C05485=1219.742,-85.560,-37.736,179.582,5.371,149.062
C05486=1219.736,-85.310,-37.746,179.584,5.371,149.061
C05487=1219.731,-85.061,-37.758,179.587,5.372,149.061
C05488=1219.726,-84.810,-37.768,179.589,5.371,149.060
C05489=1219.721,-84.561,-37.779,179.592,5.372,149.059
C05490=1219.715,-84.311,-37.790,179.594,5.371,149.058
C05491=1219.711,-84.061,-37.802,179.596,5.372,149.058
C05492=1219.705,-83.812,-37.813,179.599,5.372,149.057
C05493=1219.700,-83.562,-37.823,179.601,5.372,149.056
C05494=1219.696,-83.312,-37.834,179.603,5.372,149.056
C05495=1219.689,-83.063,-37.845,179.606,5.372,149.055
C05496=1219.685,-82.813,-37.857,179.608,5.372,149.054
C05497=1219.680,-82.563,-37.868,179.610,5.373,149.054
C05498=1219.674,-82.314,-37.878,179.612,5.372,149.053
C05499=1219.669,-82.064,-37.890,179.615,5.373,149.052
C05500=1219.664,-81.814,-37.901,179.617,5.372,149.052
C05501=1219.659,-81.565,-37.911,179.620,5.373,149.051
C05502=1219.653,-81.315,-37.923,179.622,5.372,149.050
C05503=1219.648,-81.064,-37.934,179.625,5.373,149.049
C05504=1219.643,-80.816,-37.945,179.627,5.372,149.049
C05505=1219.638,-80.566,-37.956,179.629,5.373,149.048
C05506=1219.632,-80.315,-37.967,179.632,5.374,149.048
C05507=1219.627,-80.066,-37.978,179.634,5.373,149.047
C05508=1219.622,-79.817,-37.990,179.636,5.374,149.046
C05509=1219.617,-79.567,-38.001,179.638,5.373,149.045
C05510=1219.612,-79.317,-38.012,179.641,5.374,149.045
C05511=1219.607,-79.068,-38.023,179.643,5.374,149.044
C05512=1219.601,-78.818,-38.035,179.646,5.374,149.043
C05513=1219.596,-78.568,-38.045,179.648,5.374,149.043
C05514=1219.591,-78.319,-38.056,179.651,5.374,149.042
C05515=1219.586,-78.069,-38.068,179.653,5.374,149.041
C05516=1219.581,-77.819,-38.079,179.655,5.374,149.041
C05517=1219.576,-77.569,-38.090,179.657,5.374,149.040
C05518=1219.570,-77.320,-38.102,179.660,5.375,149.039
C05519=1219.565,-77.070,-38.113,179.662,5.374,149.039
C05520=1219.561,-76.820,-38.124,179.664,5.375,149.038
C05521=1219.554,-76.571,-38.136,179.667,5.375,149.037
C05522=1219.549,-76.321,-38.146,179.669,5.375,149.036
C05523=1219.544,-76.071,-38.158,179.672,5.375,149.036
C05524=1219.539,-75.821,-38.169,179.674,5.375,149.035
C05525=1219.534,-75.572,-38.180,179.677,5.375,149.034
C05526=1219.529,-75.322,-38.192,179.679,5.375,149.034
C05527=1219.523,-75.051,-38.204,179.681,5.375,149.033
C05528=1219.517,-74.781,-38.216,179.684,5.376,149.032
C05529=1219.512,-74.511,-38.229,179.686,5.376,149.032
C05530=1219.507,-74.240,-38.241,179.689,5.376,149.031
C05531=1219.501,-73.991,-38.253,179.691,5.376,149.030
C05532=1219.496,-73.741,-38.264,179.693,5.376,149.029
C05533=1219.490,-73.491,-38.276,179.696,5.377,149.029
C05534=1219.485,-73.241,-38.286,179.698,5.376,149.028
C05535=1219.480,-72.991,-38.298,179.701,5.377,149.027
C05536=1219.475,-72.742,-38.309,179.703,5.376,149.027
C05537=1219.470,-72.493,-38.320,179.706,5.377,149.026
C05538=1219.465,-72.243,-38.332,179.708,5.376,149.025
C05539=1219.460,-71.993,-38.344,179.710,5.377,149.024
C05540=1219.454,-71.743,-38.355,179.713,5.377,149.024
C05541=1219.449,-71.494,-38.366,179.715,5.377,149.023
C05542=1219.444,-71.244,-38.378,179.718,5.377,149.022
C05543=1219.439,-70.995,-38.390,179.720,5.377,149.022
C05544=1219.434,-70.745,-38.401,179.723,5.378,149.021
C05545=1219.429,-70.495,-38.413,179.724,5.378,149.020
C05546=1219.423,-70.246,-38.424,179.727,5.378,149.020
C05547=1219.418,-69.996,-38.435,179.729,5.378,149.019
C05548=1219.413,-69.746,-38.447,179.732,5.378,149.018
C05549=1219.408,-69.496,-38.458,179.734,5.378,149.018
C05550=1219.402,-69.246,-38.470,179.736,5.378,149.017
C05551=1219.398,-68.996,-38.481,179.739,5.379,149.016
C05552=1219.392,-68.747,-38.493,179.741,5.378,149.015
C05553=1219.386,-68.497,-38.505,179.744,5.379,149.015
C05554=1219.382,-68.248,-38.516,179.746,5.378,149.014
C05555=1219.376,-67.998,-38.528,179.749,5.379,149.013
C05556=1219.372,-67.749,-38.540,179.751,5.379,149.013
C05557=1219.366,-67.499,-38.552,179.753,5.379,149.012
C05558=1219.362,-67.249,-38.563,179.755,5.379,149.011
C05559=1219.356,-67.000,-38.574,179.758,5.379,149.011
C05560=1219.351,-66.750,-38.586,179.760,5.380,149.010
C05561=1219.345,-66.500,-38.598,179.762,5.380,149.009
C05562=1219.340,-66.250,-38.609,179.765,5.380,149.009
C05563=1219.335,-66.001,-38.621,179.767,5.380,149.008
C05564=1219.330,-65.751,-38.633,179.770,5.380,149.007
C05565=1219.325,-65.501,-38.644,179.772,5.380,149.007
C05566=1219.320,-65.251,-38.656,179.775,5.380,149.006
C05567=1219.314,-65.001,-38.668,179.777,5.381,149.005
C05568=1219.309,-64.752,-38.679,179.779,5.380,149.004
C05569=1219.304,-64.503,-38.691,179.782,5.381,149.004
C05570=1219.299,-64.254,-38.703,179.784,5.381,149.003
C05571=1219.294,-64.004,-38.714,179.787,5.381,149.002
C05572=1219.288,-63.754,-38.726,179.789,5.381,149.002
C05573=1219.284,-63.504,-38.738,179.791,5.381,149.001
C05574=1219.278,-63.254,-38.749,179.794,5.382,149.000
C05575=1219.273,-63.005,-38.762,179.796,5.381,148.999
C05576=1219.268,-62.755,-38.773,179.799,5.382,148.999
C05577=1219.263,-62.505,-38.785,179.801,5.381,148.998
C05578=1219.258,-62.255,-38.797,179.803,5.382,148.998
C05579=1219.253,-62.006,-38.808,179.805,5.382,148.997
C05580=1219.247,-61.756,-38.820,179.808,5.382,148.996
C05581=1219.242,-61.507,-38.833,179.811,5.383,148.995
C05582=1219.237,-61.257,-38.844,179.813,5.382,148.995
C05583=1219.232,-61.008,-38.856,179.815,5.383,148.994
C05584=1219.226,-60.758,-38.868,179.817,5.383,148.993
C05585=1219.222,-60.509,-38.880,179.820,5.383,148.993
C05586=1219.216,-60.259,-38.891,179.822,5.383,148.992
C05587=1219.211,-60.009,-38.903,179.825,5.383,148.991
C05588=1219.206,-59.759,-38.915,179.828,5.384,148.991
C05589=1219.201,-59.510,-38.927,179.830,5.383,148.990
C05590=1219.196,-59.260,-38.939,179.832,5.384,148.989
C05591=1219.190,-59.010,-38.951,179.834,5.383,148.988
C05592=1219.186,-58.761,-38.963,179.837,5.384,148.988
C05593=1219.180,-58.511,-38.975,179.840,5.384,148.987
C05594=1219.175,-58.261,-38.987,179.842,5.384,148.986
C05595=1219.170,-58.011,-38.999,179.844,5.384,148.986
C05596=1219.165,-57.762,-39.011,179.847,5.384,148.985
C05597=1219.160,-57.512,-39.023,179.849,5.385,148.984
C05598=1219.154,-57.262,-39.034,179.851,5.385,148.984
C05599=1219.149,-57.013,-39.047,179.853,5.385,148.983
C05600=1219.145,-56.763,-39.058,179.856,5.385,148.982
C05601=1219.139,-56.514,-39.071,179.858,5.385,148.982
C05602=1219.134,-56.264,-39.083,179.861,5.386,148.981
C05603=1219.129,-56.014,-39.095,179.863,5.385,148.980
C05604=1219.123,-55.765,-39.107,179.866,5.386,148.979
C05605=1219.119,-55.515,-39.119,179.868,5.386,148.979
C05606=1219.113,-55.265,-39.131,179.870,5.386,148.978
C05607=1219.108,-55.016,-39.143,179.873,5.386,148.977
C05608=1219.103,-54.766,-39.155,179.875,5.386,148.977
C05609=1219.098,-54.517,-39.168,179.878,5.386,148.976
C05610=1219.093,-54.267,-39.179,179.880,5.387,148.975
C05611=1219.088,-54.016,-39.191,179.883,5.387,148.975
C05612=1219.083,-53.767,-39.204,179.885,5.387,148.974
C05613=1219.078,-53.517,-39.216,179.887,5.387,148.973
C05614=1219.072,-53.268,-39.228,179.890,5.387,148.972
C05615=1219.067,-53.018,-39.240,179.893,5.388,148.972
C05616=1219.063,-52.769,-39.252,179.895,5.387,148.971
C05617=1219.057,-52.519,-39.264,179.897,5.388,148.970
C05618=1219.052,-52.270,-39.277,179.899,5.387,148.970
C05619=1219.047,-52.020,-39.288,179.902,5.388,148.969
C05620=1219.042,-51.770,-39.301,179.904,5.389,148.968
C05621=1219.036,-51.520,-39.313,179.906,5.388,148.968
C05622=1219.031,-51.271,-39.326,179.909,5.389,148.967
C05623=1219.026,-51.021,-39.337,179.911,5.389,148.966
C05624=1219.021,-50.772,-39.349,179.914,5.389,148.966
C05625=1219.016,-50.521,-39.362,179.916,5.389,148.965
C05626=1219.011,-50.272,-39.374,179.919,5.389,148.964
C05627=1219.006,-50.022,-39.386,179.921,5.390,148.964
C05628=1219.001,-49.773,-39.399,179.924,5.390,148.963
C05629=1218.995,-49.523,-39.411,179.926,5.390,148.962
C05630=1218.990,-49.274,-39.423,179.929,5.390,148.961
C05631=1218.985,-49.003,-39.436,179.931,5.390,148.961
C05632=1218.979,-48.734,-39.450,179.933,5.390,148.960
C05633=1218.973,-48.464,-39.463,179.937,5.390,148.959
C05634=1218.968,-48.194,-39.477,179.939,5.391,148.958
C05635=1218.963,-47.944,-39.489,179.941,5.391,148.958
C05636=1218.958,-47.695,-39.501,179.944,5.391,148.957
C05637=1218.952,-47.445,-39.514,179.947,5.392,148.956
C05638=1218.947,-47.195,-39.526,179.949,5.391,148.956
C05639=1218.942,-46.946,-39.538,179.951,5.392,148.955
C05640=1218.937,-46.696,-39.551,179.953,5.391,148.954
C05641=1218.932,-46.446,-39.563,179.956,5.392,148.953
C05642=1218.927,-46.197,-39.576,179.959,5.392,148.953
C05643=1218.922,-45.947,-39.588,179.960,5.392,148.952
C05644=1218.916,-45.698,-39.600,179.963,5.393,148.952
C05645=1218.911,-45.448,-39.613,179.966,5.393,148.951
C05646=1218.906,-45.199,-39.626,179.968,5.393,148.950
C05647=1218.901,-44.948,-39.638,179.970,5.393,148.949
C05648=1218.896,-44.699,-39.650,179.973,5.393,148.949
C05649=1218.891,-44.450,-39.663,179.975,5.394,148.948
C05650=1218.886,-44.200,-39.675,179.978,5.394,148.947
C05651=1218.880,-43.950,-39.687,179.980,5.394,148.947
C05652=1218.876,-43.700,-39.700,179.983,5.394,148.946
C05653=1218.871,-43.451,-39.713,179.985,5.395,148.945
C05654=1218.865,-43.201,-39.725,179.987,5.394,148.945
C05655=1218.860,-42.952,-39.738,179.990,5.395,148.944
C05656=1218.855,-42.702,-39.750,179.992,5.394,148.943
C05657=1218.851,-42.452,-39.763,179.995,5.395,148.942
C05658=1218.845,-42.203,-39.775,179.997,5.395,148.942
C05659=1218.839,-41.953,-39.788,180.000,5.395,148.941
C05660=1218.834,-41.704,-39.801,-179.998,5.396,148.940
C05661=1218.829,-41.454,-39.813,-179.995,5.396,148.940
C05662=1218.824,-41.204,-39.826,-179.993,5.396,148.939
C05663=1218.819,-40.954,-39.838,-179.990,5.396,148.938
C05664=1218.814,-40.705,-39.851,-179.988,5.397,148.938
C05665=1218.809,-40.456,-39.863,-179.986,5.396,148.937
C05666=1218.804,-40.206,-39.876,-179.983,5.397,148.936
C05667=1218.799,-39.956,-39.889,-179.981,5.397,148.935
C05668=1218.793,-39.707,-39.902,-179.978,5.397,148.935
C05669=1218.788,-39.457,-39.914,-179.976,5.398,148.934
C05670=1218.783,-39.207,-39.927,-179.974,5.398,148.934
C05671=1218.778,-38.957,-39.940,-179.971,5.398,148.933
C05672=1218.773,-38.708,-39.952,-179.969,5.398,148.932
C05673=1218.768,-38.459,-39.965,-179.967,5.398,148.931
C05674=1218.763,-38.209,-39.978,-179.964,5.399,148.931
C05675=1218.758,-37.959,-39.991,-179.961,5.399,148.930
C05676=1218.752,-37.710,-40.004,-179.959,5.399,148.929
C05677=1218.747,-37.460,-40.015,-179.957,5.399,148.929
C05678=1218.743,-37.210,-40.028,-179.954,5.400,148.928
C05679=1218.737,-36.961,-40.041,-179.952,5.399,148.927
C05680=1218.732,-36.711,-40.054,-179.949,5.400,148.927
C05681=1218.727,-36.461,-40.067,-179.947,5.400,148.926
C05682=1218.722,-36.212,-40.080,-179.944,5.400,148.925
C05683=1218.717,-35.962,-40.092,-179.942,5.401,148.924
C05684=1218.712,-35.713,-40.105,-179.940,5.400,148.924
C05685=1218.706,-35.463,-40.119,-179.937,5.401,148.923
C05686=1218.701,-35.213,-40.131,-179.934,5.401,148.922
C05687=1218.696,-34.964,-40.144,-179.932,5.401,148.922
C05688=1218.692,-34.714,-40.157,-179.930,5.401,148.921
C05689=1218.686,-34.464,-40.170,-179.927,5.402,148.920
C05690=1218.681,-34.215,-40.183,-179.925,5.402,148.920
C05691=1218.676,-33.965,-40.196,-179.922,5.402,148.919
C05692=1218.671,-33.716,-40.208,-179.919,5.402,148.918
C05693=1218.665,-33.466,-40.221,-179.917,5.402,148.917
C05694=1218.661,-33.216,-40.234,-179.915,5.403,148.917
C05695=1218.655,-32.967,-40.247,-179.912,5.403,148.916
C05696=1218.650,-32.717,-40.259,-179.910,5.403,148.916
C05697=1218.645,-32.467,-40.273,-179.908,5.404,148.915
C05698=1218.640,-32.218,-40.286,-179.905,5.404,148.914
C05699=1218.635,-31.968,-40.298,-179.903,5.404,148.914
C05700=1218.630,-31.718,-40.312,-179.900,5.404,148.913
C05701=1218.625,-31.469,-40.325,-179.898,5.405,148.912
C05702=1218.620,-31.220,-40.338,-179.896,5.404,148.911
C05703=1218.614,-30.970,-40.351,-179.893,5.405,148.911
C05704=1218.609,-30.720,-40.364,-179.890,5.405,148.910
C05705=1218.605,-30.470,-40.377,-179.888,5.405,148.909
C05706=1218.599,-30.221,-40.390,-179.886,5.406,148.909
C05707=1218.594,-29.971,-40.403,-179.883,5.406,148.908
C05708=1218.589,-29.721,-40.416,-179.881,5.406,148.907
C05709=1218.584,-29.472,-40.430,-179.878,5.406,148.907
C05710=1218.579,-29.223,-40.442,-179.876,5.407,148.906
C05711=1218.574,-28.973,-40.455,-179.873,5.406,148.905
C05712=1218.568,-28.723,-40.468,-179.871,5.407,148.904
C05713=1218.564,-28.473,-40.481,-179.868,5.407,148.904
C05714=1218.559,-28.224,-40.494,-179.866,5.407,148.903
C05715=1218.554,-27.974,-40.508,-179.863,5.408,148.902
C05716=1218.548,-27.725,-40.521,-179.861,5.408,148.902
C05717=1218.543,-27.475,-40.534,-179.859,5.408,148.901
C05718=1218.538,-27.225,-40.547,-179.856,5.408,148.900
C05719=1218.533,-26.976,-40.559,-179.853,5.409,148.900
C05720=1218.528,-26.726,-40.574,-179.851,5.409,148.899
C05721=1218.523,-26.477,-40.586,-179.849,5.409,148.898
C05722=1218.517,-26.228,-40.600,-179.846,5.409,148.897
C05723=1218.512,-25.977,-40.613,-179.843,5.410,148.897
C05724=1218.508,-25.729,-40.626,-179.842,5.410,148.896
C05725=1218.502,-25.478,-40.639,-179.839,5.410,148.896
C05726=1218.497,-25.229,-40.652,-179.836,5.411,148.895
C05727=1218.492,-24.979,-40.666,-179.834,5.411,148.894
C05728=1218.487,-24.730,-40.679,-179.832,5.411,148.894
C05729=1218.482,-24.480,-40.692,-179.829,5.412,148.893
C05730=1218.477,-24.230,-40.705,-179.827,5.411,148.892
C05731=1218.472,-23.981,-40.719,-179.824,5.412,148.891
C05732=1218.467,-23.731,-40.732,-179.822,5.412,148.891
C05733=1218.461,-23.481,-40.745,-179.819,5.412,148.890
C05734=1218.457,-23.232,-40.759,-179.817,5.412,148.889
C05735=1218.451,-22.962,-40.773,-179.814,5.413,148.889
C05736=1218.446,-22.694,-40.787,-179.811,5.413,148.888
C05737=1218.440,-22.424,-40.801,-179.808,5.414,148.887
C05738=1218.434,-22.155,-40.816,-179.806,5.414,148.886
C05739=1218.429,-21.905,-40.829,-179.804,5.414,148.886
C05740=1218.424,-21.655,-40.843,-179.801,5.414,148.885
C05741=1218.419,-21.406,-40.856,-179.798,5.415,148.884
C05742=1218.414,-21.156,-40.870,-179.796,5.414,148.884
C05743=1218.409,-20.907,-40.883,-179.794,5.415,148.883
C05744=1218.404,-20.657,-40.896,-179.791,5.415,148.882
C05745=1218.399,-20.408,-40.910,-179.789,5.415,148.881
C05746=1218.394,-20.158,-40.923,-179.786,5.416,148.881
C05747=1218.389,-19.908,-40.937,-179.783,5.416,148.880
C05748=1218.384,-19.659,-40.950,-179.781,5.417,148.880
C05749=1218.379,-19.409,-40.964,-179.779,5.417,148.879
C05750=1218.374,-19.160,-40.977,-179.777,5.417,148.878
C05751=1218.369,-18.910,-40.991,-179.774,5.418,148.878
C05752=1218.364,-18.661,-41.004,-179.772,5.417,148.877
C05753=1218.358,-18.410,-41.017,-179.769,5.418,148.876
C05754=1218.353,-18.161,-41.031,-179.767,5.418,148.875
C05755=1218.348,-17.911,-41.044,-179.764,5.419,148.875
C05756=1218.343,-17.662,-41.058,-179.762,5.418,148.874
C05757=1218.338,-17.413,-41.072,-179.759,5.419,148.873
C05758=1218.333,-17.163,-41.085,-179.756,5.419,148.873
C05759=1218.328,-16.914,-41.099,-179.754,5.419,148.872
C05760=1218.323,-16.664,-41.112,-179.752,5.420,148.871
C05761=1218.318,-16.415,-41.126,-179.749,5.420,148.871
C05762=1218.312,-16.164,-41.140,-179.746,5.421,148.870
C05763=1218.307,-15.916,-41.153,-179.744,5.420,148.869
C05764=1218.302,-15.665,-41.167,-179.742,5.421,148.869
C05765=1218.297,-15.415,-41.181,-179.739,5.421,148.868
C05766=1218.292,-15.166,-41.194,-179.737,5.421,148.867
C05767=1218.287,-14.916,-41.208,-179.734,5.422,148.866
C05768=1218.282,-14.667,-41.222,-179.732,5.422,148.866
C05769=1218.277,-14.417,-41.235,-179.729,5.423,148.865
C05770=1218.272,-14.168,-41.249,-179.727,5.422,148.864
C05771=1218.267,-13.919,-41.263,-179.725,5.423,148.864
C05772=1218.262,-13.669,-41.276,-179.722,5.424,148.863
C05773=1218.257,-13.420,-41.290,-179.719,5.424,148.862
C05774=1218.251,-13.169,-41.303,-179.717,5.424,148.862
C05775=1218.247,-12.920,-41.317,-179.715,5.424,148.861
C05776=1218.241,-12.671,-41.331,-179.712,5.425,148.860
C05777=1218.236,-12.421,-41.344,-179.710,5.424,148.860
C05778=1218.231,-12.171,-41.359,-179.707,5.425,148.859
C05779=1218.226,-11.922,-41.372,-179.705,5.425,148.858
C05780=1218.221,-11.672,-41.386,-179.702,5.426,148.858
C05781=1218.216,-11.423,-41.400,-179.700,5.426,148.857
C05782=1218.211,-11.173,-41.413,-179.697,5.426,148.856
C05783=1218.206,-10.924,-41.427,-179.695,5.427,148.856
C05784=1218.201,-10.674,-41.441,-179.692,5.427,148.855
C05785=1218.196,-10.424,-41.455,-179.690,5.427,148.854
C05786=1218.191,-10.175,-41.469,-179.687,5.427,148.853
C05787=1218.186,-9.926,-41.483,-179.685,5.428,148.853
C05788=1218.181,-9.676,-41.496,-179.682,5.428,148.852
C05789=1218.176,-9.426,-41.510,-179.680,5.428,148.851
C05790=1218.170,-9.177,-41.524,-179.677,5.429,148.851
C05791=1218.166,-8.928,-41.538,-179.674,5.429,148.850
C05792=1218.161,-8.677,-41.552,-179.672,5.430,148.850
C05793=1218.156,-8.428,-41.566,-179.670,5.430,148.849
C05794=1218.150,-8.179,-41.580,-179.668,5.430,148.848
C05795=1218.145,-7.929,-41.594,-179.665,5.431,148.847
C05796=1218.141,-7.679,-41.608,-179.662,5.431,148.847
C05797=1218.135,-7.430,-41.621,-179.660,5.431,148.846
C05798=1218.130,-7.180,-41.635,-179.658,5.431,148.845
C05799=1218.125,-6.930,-41.649,-179.655,5.432,148.845
C05800=1218.120,-6.681,-41.663,-179.652,5.432,148.844
C05801=1218.115,-6.432,-41.678,-179.650,5.432,148.843
C05802=1218.110,-6.182,-41.691,-179.648,5.433,148.843
C05803=1218.105,-5.933,-41.706,-179.645,5.433,148.842
C05804=1218.100,-5.683,-41.719,-179.642,5.434,148.841
C05805=1218.095,-5.433,-41.733,-179.640,5.433,148.841
C05806=1218.090,-5.183,-41.747,-179.637,5.434,148.840
C05807=1218.085,-4.934,-41.762,-179.635,5.434,148.839
C05808=1218.079,-4.685,-41.776,-179.632,5.435,148.839
C05809=1218.074,-4.435,-41.790,-179.630,5.435,148.838
C05810=1218.070,-4.186,-41.803,-179.627,5.435,148.837
C05811=1218.065,-3.936,-41.818,-179.625,5.436,148.837
C05812=1218.060,-3.687,-41.832,-179.623,5.436,148.836
C05813=1218.055,-3.437,-41.846,-179.621,5.436,148.835
C05814=1218.050,-3.188,-41.860,-179.618,5.437,148.835
C05815=1218.045,-2.938,-41.875,-179.615,5.437,148.834
C05816=1218.039,-2.689,-41.888,-179.613,5.438,148.833
C05817=1218.034,-2.438,-41.902,-179.610,5.438,148.833
C05818=1218.029,-2.189,-41.916,-179.608,5.438,148.832
C05819=1218.024,-1.939,-41.931,-179.605,5.438,148.831
C05820=1218.019,-1.689,-41.945,-179.603,5.439,148.830
C05821=1218.013,-1.440,-41.959,-179.600,5.439,148.830
C05822=1218.009,-1.191,-41.974,-179.598,5.439,148.829
C05823=1218.004,-0.942,-41.988,-179.595,5.440,148.828
C05824=1217.999,-0.692,-42.002,-179.593,5.440,148.828
C05825=1217.994,-0.442,-42.017,-179.590,5.441,148.827
C05826=1217.988,-0.193,-42.030,-179.587,5.441,148.826
C05827=1217.983,0.057,-42.045,-179.585,5.441,148.826
C05828=1217.978,0.306,-42.059,-179.583,5.442,148.825
C05829=1217.973,0.556,-42.073,-179.580,5.442,148.824
C05830=1217.969,0.806,-42.088,-179.578,5.443,148.824
C05831=1217.963,1.055,-42.101,-179.576,5.442,148.823
C05832=1217.958,1.304,-42.116,-179.573,5.443,148.822
C05833=1217.953,1.554,-42.130,-179.570,5.444,148.822
C05834=1217.948,1.804,-42.144,-179.568,5.444,148.821
C05835=1217.943,2.054,-42.159,-179.565,5.445,148.820
C05836=1217.939,2.303,-42.174,-179.563,5.444,148.820
C05837=1217.933,2.552,-42.187,-179.560,5.445,148.819
C05838=1217.928,2.801,-42.202,-179.558,5.445,148.818
C05839=1217.923,3.071,-42.217,-179.555,5.446,148.818
C05840=1217.917,3.340,-42.232,-179.552,5.446,148.817
C05841=1217.912,3.608,-42.248,-179.550,5.447,148.816
C05842=1217.906,3.878,-42.264,-179.546,5.447,148.815
C05843=1217.901,4.127,-42.279,-179.544,5.448,148.815
C05844=1217.897,4.377,-42.293,-179.542,5.448,148.814
C05845=1217.891,4.626,-42.307,-179.540,5.448,148.813
C05846=1217.886,4.876,-42.321,-179.537,5.449,148.813
C05847=1217.881,5.125,-42.335,-179.534,5.449,148.812
C05848=1217.876,5.374,-42.350,-179.532,5.450,148.811
C05849=1217.871,5.624,-42.365,-179.530,5.449,148.811
C05850=1217.867,5.874,-42.379,-179.527,5.450,148.810
C05851=1217.861,6.124,-42.394,-179.524,5.450,148.809
C05852=1217.856,6.373,-42.409,-179.522,5.451,148.809
C05853=1217.851,6.623,-42.423,-179.519,5.451,148.808
C05854=1217.846,6.872,-42.437,-179.517,5.451,148.807
C05855=1217.841,7.121,-42.451,-179.514,5.452,148.807
C05856=1217.836,7.371,-42.466,-179.512,5.452,148.806
C05857=1217.831,7.620,-42.481,-179.509,5.453,148.805
C05858=1217.825,7.870,-42.496,-179.507,5.454,148.805
C05859=1217.821,8.119,-42.511,-179.505,5.453,148.804
C05860=1217.816,8.369,-42.525,-179.502,5.454,148.803
C05861=1217.811,8.619,-42.539,-179.499,5.454,148.803
C05862=1217.806,8.868,-42.554,-179.497,5.455,148.802
C05863=1217.801,9.118,-42.568,-179.494,5.455,148.801
C05864=1217.796,9.368,-42.583,-179.491,5.456,148.801
C05865=1217.791,9.617,-42.598,-179.489,5.456,148.800
C05866=1217.786,9.866,-42.612,-179.487,5.456,148.799
C05867=1217.781,10.116,-42.627,-179.484,5.457,148.799
C05868=1217.776,10.366,-42.642,-179.481,5.457,148.798
C05869=1217.771,10.615,-42.657,-179.479,5.458,148.797
C05870=1217.766,10.864,-42.672,-179.477,5.458,148.797
C05871=1217.761,11.114,-42.686,-179.475,5.458,148.796
C05872=1217.756,11.364,-42.700,-179.472,5.459,148.795
C05873=1217.751,11.613,-42.716,-179.469,5.459,148.795
C05874=1217.746,11.863,-42.730,-179.467,5.460,148.794
C05875=1217.741,12.112,-42.745,-179.464,5.460,148.793
C05876=1217.735,12.362,-42.760,-179.462,5.460,148.793
C05877=1217.731,12.611,-42.775,-179.459,5.461,148.792
C05878=1217.726,12.861,-42.789,-179.457,5.461,148.791
C05879=1217.721,13.110,-42.803,-179.454,5.462,148.791
C05880=1217.715,13.360,-42.819,-179.451,5.462,148.790
C05881=1217.711,13.610,-42.833,-179.449,5.463,148.789
C05882=1217.706,13.859,-42.848,-179.447,5.463,148.789
C05883=1217.700,14.109,-42.863,-179.444,5.463,148.788
C05884=1217.696,14.358,-42.878,-179.442,5.464,148.787
C05885=1217.691,14.607,-42.892,-179.439,5.464,148.787
C05886=1217.685,14.857,-42.908,-179.436,5.465,148.786
C05887=1217.681,15.106,-42.923,-179.434,5.465,148.785
C05888=1217.676,15.356,-42.937,-179.432,5.465,148.785
C05889=1217.670,15.605,-42.953,-179.429,5.466,148.784
C05890=1217.665,15.855,-42.967,-179.426,5.466,148.783
C05891=1217.661,16.104,-42.982,-179.424,5.467,148.783
C05892=1217.655,16.354,-42.997,-179.421,5.467,148.782
C05893=1217.650,16.603,-43.012,-179.418,5.468,148.781
C05894=1217.645,16.853,-43.026,-179.416,5.469,148.781
C05895=1217.640,17.102,-43.042,-179.414,5.468,148.780
C05896=1217.635,17.351,-43.057,-179.412,5.469,148.779
C05897=1217.630,17.601,-43.071,-179.409,5.469,148.779
C05898=1217.625,17.850,-43.087,-179.406,5.470,148.778
C05899=1217.620,18.099,-43.102,-179.404,5.470,148.777
C05900=1217.615,18.350,-43.117,-179.401,5.471,148.777
C05901=1217.611,18.599,-43.132,-179.398,5.471,148.776
C05902=1217.606,18.849,-43.146,-179.396,5.471,148.775
C05903=1217.600,19.098,-43.162,-179.394,5.472,148.775
C05904=1217.596,19.347,-43.177,-179.392,5.473,148.774
C05905=1217.590,19.597,-43.192,-179.389,5.473,148.774
C05906=1217.585,19.847,-43.207,-179.386,5.474,148.773
C05907=1217.580,20.096,-43.222,-179.384,5.474,148.772
C05908=1217.575,20.345,-43.237,-179.381,5.475,148.772
C05909=1217.569,20.595,-43.252,-179.379,5.474,148.771
C05910=1217.565,20.845,-43.267,-179.376,5.475,148.770
C05911=1217.561,21.094,-43.282,-179.374,5.476,148.769
C05912=1217.555,21.344,-43.297,-179.371,5.476,148.769
C05913=1217.550,21.593,-43.312,-179.368,5.477,148.768
C05914=1217.545,21.842,-43.328,-179.366,5.477,148.768
C05915=1217.540,22.092,-43.343,-179.363,5.478,148.767
C05916=1217.535,22.342,-43.358,-179.361,5.479,148.766
C05917=1217.531,22.591,-43.373,-179.359,5.478,148.766
C05918=1217.525,22.841,-43.389,-179.356,5.479,148.765
C05919=1217.521,23.090,-43.404,-179.353,5.479,148.764
C05920=1217.515,23.339,-43.419,-179.351,5.480,148.764
C05921=1217.510,23.589,-43.434,-179.348,5.480,148.763
C05922=1217.505,23.838,-43.449,-179.346,5.481,148.762
C05923=1217.499,24.088,-43.465,-179.343,5.481,148.762
C05924=1217.495,24.338,-43.480,-179.341,5.482,148.761
C05925=1217.490,24.587,-43.496,-179.339,5.482,148.760
C05926=1217.485,24.836,-43.511,-179.336,5.483,148.760
C05927=1217.480,25.086,-43.526,-179.333,5.483,148.759
C05928=1217.475,25.335,-43.541,-179.331,5.484,148.758
C05929=1217.470,25.585,-43.557,-179.328,5.484,148.758
C05930=1217.466,25.834,-43.572,-179.325,5.485,148.757
C05931=1217.460,26.084,-43.587,-179.323,5.485,148.756
C05932=1217.455,26.333,-43.603,-179.320,5.486,148.756
C05933=1217.450,26.582,-43.618,-179.318,5.487,148.755
C05934=1217.445,26.832,-43.634,-179.316,5.486,148.754
C05935=1217.441,27.081,-43.649,-179.313,5.487,148.754
C05936=1217.435,27.331,-43.664,-179.311,5.487,148.753
C05937=1217.430,27.581,-43.679,-179.308,5.488,148.752
C05938=1217.425,27.830,-43.694,-179.305,5.489,148.752
C05939=1217.420,28.080,-43.710,-179.303,5.489,148.751
C05940=1217.416,28.329,-43.725,-179.300,5.490,148.750
C05941=1217.410,28.579,-43.741,-179.298,5.491,148.750
C05942=1217.405,28.828,-43.756,-179.295,5.491,148.749
C05943=1217.400,29.096,-43.773,-179.293,5.492,148.749
C05944=1217.395,29.365,-43.790,-179.289,5.492,148.748
C05945=1217.389,29.634,-43.806,-179.287,5.492,148.747
C05946=1217.384,29.903,-43.823,-179.284,5.493,148.746
C05947=1217.379,30.152,-43.838,-179.282,5.493,148.746
C05948=1217.374,30.401,-43.854,-179.279,5.494,148.745
C05949=1217.369,30.652,-43.870,-179.277,5.495,148.745
C05950=1217.364,30.901,-43.885,-179.275,5.495,148.744
C05951=1217.359,31.150,-43.900,-179.272,5.495,148.743
C05952=1217.353,31.399,-43.916,-179.269,5.496,148.743
C05953=1217.349,31.649,-43.931,-179.267,5.496,148.742
C05954=1217.344,31.899,-43.947,-179.264,5.497,148.741
C05955=1217.339,32.147,-43.963,-179.261,5.497,148.740
C05956=1217.334,32.397,-43.979,-179.259,5.498,148.740
C05957=1217.329,32.647,-43.994,-179.257,5.499,148.739
C05958=1217.324,32.896,-44.010,-179.254,5.499,148.739
C05959=1217.319,33.145,-44.025,-179.251,5.500,148.738
C05960=1217.314,33.395,-44.041,-179.249,5.500,148.737
C05961=1217.309,33.645,-44.056,-179.246,5.501,148.737
C05962=1217.304,33.894,-44.072,-179.244,5.501,148.736
C05963=1217.299,34.143,-44.089,-179.241,5.501,148.735
C05964=1217.294,34.393,-44.104,-179.239,5.502,148.735
C05965=1217.289,34.642,-44.119,-179.237,5.503,148.734
C05966=1217.285,34.892,-44.135,-179.234,5.503,148.734
C05967=1217.279,35.141,-44.151,-179.231,5.504,148.733
C05968=1217.274,35.391,-44.166,-179.229,5.504,148.732
C05969=1217.269,35.640,-44.183,-179.226,5.505,148.731
C05970=1217.265,35.889,-44.198,-179.223,5.505,148.731
C05971=1217.259,36.139,-44.214,-179.221,5.506,148.730
C05972=1217.254,36.389,-44.230,-179.219,5.507,148.730
C05973=1217.249,36.638,-44.246,-179.216,5.507,148.729
C05974=1217.245,36.888,-44.262,-179.213,5.508,148.728
C05975=1217.239,37.137,-44.277,-179.211,5.508,148.728
C05976=1217.235,37.386,-44.292,-179.208,5.509,148.727
C05977=1217.230,37.636,-44.309,-179.206,5.509,148.726
C05978=1217.225,37.885,-44.325,-179.203,5.509,148.726
C05979=1217.219,38.135,-44.340,-179.201,5.510,148.725
C05980=1217.215,38.385,-44.356,-179.198,5.511,148.725
C05981=1217.209,38.634,-44.372,-179.196,5.511,148.724
C05982=1217.205,38.884,-44.388,-179.193,5.512,148.723
C05983=1217.200,39.133,-44.403,-179.191,5.512,148.722
C05984=1217.195,39.381,-44.420,-179.188,5.513,148.722
C05985=1217.190,39.632,-44.436,-179.186,5.514,148.721
C05986=1217.185,39.881,-44.451,-179.183,5.514,148.721
C05987=1217.180,40.130,-44.468,-179.180,5.515,148.720
C05988=1217.175,40.380,-44.484,-179.178,5.515,148.719
C05989=1217.170,40.629,-44.499,-179.175,5.516,148.719
C05990=1217.165,40.879,-44.516,-179.173,5.516,148.718
C05991=1217.160,41.128,-44.531,-179.170,5.517,148.717
C05992=1217.155,41.378,-44.548,-179.168,5.518,148.717
C05993=1217.150,41.627,-44.564,-179.165,5.518,148.716
C05994=1217.144,41.876,-44.579,-179.163,5.519,148.716
C05995=1217.140,42.126,-44.596,-179.160,5.520,148.715
C05996=1217.135,42.375,-44.611,-179.157,5.520,148.714
C05997=1217.131,42.625,-44.628,-179.155,5.521,148.714
C05998=1217.125,42.874,-44.643,-179.152,5.522,148.713
C05999=1217.121,43.123,-44.660,-179.150,5.521,148.712
C06000=1217.116,43.373,-44.675,-179.148,5.522,148.712
C06001=1217.111,43.622,-44.692,-179.145,5.522,148.711
C06002=1217.106,43.872,-44.708,-179.142,5.523,148.710
C06003=1217.101,44.121,-44.724,-179.140,5.524,148.710
C06004=1217.096,44.371,-44.740,-179.138,5.524,148.709
C06005=1217.091,44.620,-44.757,-179.135,5.525,148.709
C06006=1217.086,44.869,-44.772,-179.132,5.526,148.708
C06007=1217.081,45.118,-44.788,-179.130,5.526,148.707
C06008=1217.076,45.368,-44.804,-179.127,5.527,148.707
C06009=1217.070,45.617,-44.821,-179.124,5.527,148.706
C06010=1217.065,45.868,-44.837,-179.122,5.528,148.705
C06011=1217.060,46.116,-44.854,-179.120,5.529,148.705
C06012=1217.056,46.366,-44.870,-179.117,5.529,148.704
C06013=1217.051,46.615,-44.886,-179.114,5.530,148.703
C06014=1217.046,46.865,-44.902,-179.112,5.530,148.703
C06015=1217.041,47.115,-44.918,-179.109,5.531,148.702
C06016=1217.036,47.364,-44.935,-179.107,5.532,148.702
C06017=1217.031,47.614,-44.951,-179.104,5.532,148.701
C06018=1217.026,47.862,-44.967,-179.102,5.533,148.700
C06019=1217.022,48.113,-44.983,-179.099,5.533,148.700
C06020=1217.016,48.361,-44.999,-179.096,5.534,148.699
C06021=1217.012,48.611,-45.016,-179.094,5.535,148.698
C06022=1217.006,48.861,-45.032,-179.092,5.535,148.698
C06023=1217.001,49.110,-45.049,-179.089,5.536,148.697
C06024=1216.996,49.359,-45.065,-179.086,5.537,148.697
C06025=1216.991,49.609,-45.081,-179.084,5.537,148.696
C06026=1216.986,49.858,-45.097,-179.081,5.538,148.695
C06027=1216.982,50.107,-45.114,-179.079,5.539,148.695
C06028=1216.977,50.357,-45.130,-179.076,5.539,148.694
C06029=1216.972,50.606,-45.146,-179.074,5.540,148.693
C06030=1216.967,50.856,-45.164,-179.071,5.540,148.693
C06031=1216.962,51.105,-45.180,-179.068,5.541,148.692
C06032=1216.957,51.355,-45.196,-179.066,5.541,148.691
C06033=1216.952,51.604,-45.212,-179.064,5.542,148.691
C06034=1216.947,51.853,-45.229,-179.061,5.543,148.690
C06035=1216.943,52.103,-45.245,-179.058,5.543,148.690
C06036=1216.937,52.352,-45.262,-179.056,5.544,148.689
C06037=1216.932,52.602,-45.278,-179.053,5.544,148.688
C06038=1216.928,52.851,-45.295,-179.051,5.545,148.688
C06039=1216.923,53.100,-45.311,-179.048,5.546,148.687
C06040=1216.918,53.349,-45.328,-179.046,5.547,148.687
C06041=1216.912,53.599,-45.344,-179.043,5.547,148.686
C06042=1216.908,53.849,-45.361,-179.040,5.548,148.685
C06043=1216.903,54.098,-45.377,-179.038,5.549,148.685
C06044=1216.898,54.347,-45.394,-179.036,5.549,148.684
C06045=1216.893,54.597,-45.411,-179.033,5.550,148.683
C06046=1216.888,54.847,-45.427,-179.030,5.550,148.683
C06047=1216.883,55.115,-45.445,-179.028,5.551,148.682
C06048=1216.877,55.383,-45.463,-179.025,5.552,148.681
C06049=1216.872,55.651,-45.481,-179.022,5.553,148.681
C06050=1216.867,55.920,-45.498,-179.019,5.553,148.680
C06051=1216.861,56.170,-45.515,-179.017,5.554,148.679
C06052=1216.857,56.419,-45.532,-179.014,5.555,148.679
C06053=1216.852,56.668,-45.548,-179.012,5.555,148.678
C06054=1216.847,56.917,-45.565,-179.009,5.556,148.678
C06055=1216.842,57.167,-45.582,-179.007,5.556,148.677
C06056=1216.837,57.416,-45.599,-179.004,5.557,148.676
C06057=1216.833,57.665,-45.615,-179.002,5.558,148.676
C06058=1216.827,57.915,-45.633,-178.999,5.558,148.675
C06059=1216.822,58.164,-45.649,-178.997,5.559,148.675
C06060=1216.818,58.414,-45.666,-178.994,5.560,148.674
C06061=1216.813,58.663,-45.683,-178.991,5.560,148.673
C06062=1216.808,58.912,-45.699,-178.989,5.561,148.673
C06063=1216.803,59.162,-45.716,-178.986,5.562,148.672
C06064=1216.798,59.411,-45.733,-178.983,5.563,148.671
C06065=1216.793,59.661,-45.750,-178.981,5.564,148.671
C06066=1216.788,59.910,-45.767,-178.978,5.564,148.670
C06067=1216.783,60.159,-45.783,-178.976,5.565,148.670
C06068=1216.779,60.409,-45.800,-178.973,5.566,148.669
C06069=1216.773,60.658,-45.817,-178.971,5.566,148.668
C06070=1216.768,60.908,-45.834,-178.968,5.567,148.668
C06071=1216.763,61.157,-45.851,-178.966,5.568,148.667
C06072=1216.759,61.407,-45.867,-178.963,5.568,148.667
C06073=1216.754,61.656,-45.884,-178.961,5.569,148.666
C06074=1216.748,61.905,-45.901,-178.958,5.569,148.665
C06075=1216.744,62.155,-45.918,-178.955,5.570,148.665
C06076=1216.739,62.405,-45.935,-178.953,5.571,148.664
C06077=1216.734,62.653,-45.952,-178.951,5.571,148.663
C06078=1216.729,62.903,-45.969,-178.948,5.572,148.663
C06079=1216.724,63.152,-45.986,-178.945,5.573,148.662
C06080=1216.720,63.402,-46.003,-178.943,5.573,148.662
C06081=1216.714,63.651,-46.019,-178.940,5.575,148.661
C06082=1216.709,63.900,-46.036,-178.937,5.575,148.660
C06083=1216.704,64.150,-46.053,-178.935,5.576,148.660
C06084=1216.700,64.399,-46.071,-178.932,5.577,148.659
C06085=1216.695,64.649,-46.088,-178.930,5.578,148.659
C06086=1216.690,64.897,-46.104,-178.927,5.578,148.658
C06087=1216.684,65.147,-46.122,-178.925,5.579,148.657
C06088=1216.680,65.397,-46.138,-178.922,5.579,148.657
C06089=1216.675,65.646,-46.156,-178.920,5.580,148.656
C06090=1216.671,65.895,-46.173,-178.917,5.581,148.656
C06091=1216.665,66.144,-46.190,-178.915,5.581,148.655
C06092=1216.660,66.394,-46.207,-178.912,5.582,148.654
C06093=1216.655,66.643,-46.224,-178.910,5.583,148.654
C06094=1216.650,66.893,-46.242,-178.907,5.584,148.653
C06095=1216.646,67.142,-46.258,-178.904,5.585,148.652
C06096=1216.640,67.392,-46.276,-178.901,5.585,148.652
C06097=1216.636,67.640,-46.293,-178.899,5.586,148.651
C06098=1216.630,67.890,-46.310,-178.897,5.587,148.651
C06099=1216.626,68.140,-46.327,-178.894,5.587,148.650
C06100=1216.621,68.389,-46.345,-178.891,5.588,148.649
C06101=1216.617,68.638,-46.361,-178.889,5.589,148.649
C06102=1216.611,68.888,-46.379,-178.887,5.589,148.648
C06103=1216.606,69.137,-46.397,-178.884,5.590,148.648
C06104=1216.601,69.386,-46.413,-178.881,5.591,148.647
C06105=1216.596,69.636,-46.430,-178.879,5.592,148.647
C06106=1216.592,69.885,-46.447,-178.876,5.593,148.646
C06107=1216.587,70.135,-46.465,-178.873,5.593,148.645
C06108=1216.582,70.384,-46.483,-178.871,5.594,148.645
C06109=1216.577,70.633,-46.499,-178.869,5.595,148.644
C06110=1216.572,70.883,-46.517,-178.866,5.596,148.643
C06111=1216.567,71.132,-46.535,-178.863,5.596,148.643
C06112=1216.562,71.381,-46.551,-178.861,5.597,148.642
C06113=1216.557,71.630,-46.569,-178.859,5.598,148.642
C06114=1216.552,71.880,-46.586,-178.855,5.599,148.641
C06115=1216.548,72.129,-46.604,-178.853,5.600,148.640
C06116=1216.543,72.379,-46.621,-178.851,5.600,148.640
C06117=1216.537,72.628,-46.638,-178.848,5.601,148.639
C06118=1216.533,72.877,-46.655,-178.845,5.602,148.639
C06119=1216.528,73.127,-46.673,-178.843,5.602,148.638
C06120=1216.523,73.376,-46.691,-178.841,5.603,148.638
C06121=1216.519,73.626,-46.707,-178.838,5.604,148.637
C06122=1216.514,73.875,-46.725,-178.835,5.604,148.636
C06123=1216.508,74.125,-46.743,-178.832,5.606,148.636
C06124=1216.504,74.374,-46.761,-178.830,5.607,148.635
C06125=1216.499,74.622,-46.778,-178.827,5.607,148.635
C06126=1216.494,74.872,-46.795,-178.825,5.608,148.634
C06127=1216.489,75.121,-46.813,-178.823,5.609,148.633
C06128=1216.483,75.371,-46.830,-178.820,5.609,148.633
C06129=1216.479,75.620,-46.848,-178.817,5.610,148.632
C06130=1216.474,75.869,-46.865,-178.815,5.610,148.631
C06131=1216.469,76.119,-46.883,-178.812,5.612,148.631
C06132=1216.464,76.368,-46.901,-178.809,5.613,148.630
C06133=1216.460,76.617,-46.917,-178.807,5.613,148.630
C06134=1216.455,76.866,-46.935,-178.805,5.614,148.629
C06135=1216.450,77.116,-46.953,-178.802,5.615,148.629
C06136=1216.445,77.365,-46.971,-178.799,5.615,148.628
C06137=1216.440,77.615,-46.989,-178.797,5.616,148.627
C06138=1216.435,77.864,-47.005,-178.794,5.618,148.627
C06139=1216.430,78.113,-47.023,-178.791,5.618,148.626
C06140=1216.426,78.362,-47.041,-178.789,5.619,148.626
C06141=1216.420,78.612,-47.059,-178.787,5.620,148.625
C06142=1216.415,78.861,-47.077,-178.784,5.620,148.624
C06143=1216.410,79.111,-47.094,-178.781,5.621,148.624
C06144=1216.406,79.360,-47.111,-178.779,5.622,148.623
C06145=1216.401,79.609,-47.129,-178.776,5.623,148.623
C06146=1216.396,79.858,-47.147,-178.773,5.624,148.622
C06147=1216.391,80.108,-47.165,-178.771,5.624,148.621
C06148=1216.386,80.357,-47.182,-178.769,5.625,148.621
C06149=1216.381,80.607,-47.200,-178.766,5.626,148.620
C06150=1216.376,80.856,-47.218,-178.763,5.627,148.620
C06151=1216.371,81.124,-47.238,-178.760,5.628,148.619
C06152=1216.366,81.393,-47.256,-178.758,5.629,148.618
C06153=1216.361,81.661,-47.276,-178.755,5.629,148.618
C06154=1216.356,81.929,-47.295,-178.752,5.631,148.617
C06155=1216.350,82.179,-47.313,-178.750,5.631,148.617
C06156=1216.345,82.428,-47.330,-178.747,5.632,148.616
C06157=1216.341,82.677,-47.348,-178.745,5.633,148.616
C06158=1216.336,82.926,-47.366,-178.742,5.634,148.615
C06159=1216.331,83.176,-47.384,-178.739,5.635,148.614
C06160=1216.327,83.425,-47.402,-178.737,5.636,148.614
C06161=1216.322,83.675,-47.419,-178.734,5.636,148.613
C06162=1216.317,83.924,-47.437,-178.732,5.637,148.613
C06163=1216.312,84.174,-47.455,-178.729,5.638,148.612
C06164=1216.307,84.423,-47.473,-178.727,5.639,148.611
C06165=1216.302,84.672,-47.491,-178.724,5.640,148.611
C06166=1216.297,84.921,-47.509,-178.721,5.641,148.610
C06167=1216.292,85.170,-47.527,-178.719,5.642,148.610
C06168=1216.288,85.419,-47.545,-178.716,5.642,148.609
C06169=1216.283,85.669,-47.563,-178.714,5.643,148.608
C06170=1216.278,85.918,-47.582,-178.711,5.644,148.608
C06171=1216.273,86.168,-47.600,-178.708,5.645,148.607
C06172=1216.268,86.417,-47.618,-178.706,5.646,148.607
C06173=1216.263,86.667,-47.635,-178.704,5.647,148.606
C06174=1216.258,86.916,-47.653,-178.701,5.647,148.606
C06175=1216.253,87.165,-47.671,-178.698,5.648,148.605
C06176=1216.249,87.414,-47.689,-178.696,5.649,148.605
C06177=1216.244,87.664,-47.707,-178.693,5.650,148.604
C06178=1216.239,87.913,-47.725,-178.690,5.651,148.603
C06179=1216.234,88.163,-47.744,-178.688,5.652,148.603
C06180=1216.229,88.411,-47.762,-178.686,5.652,148.602
C06181=1216.224,88.660,-47.780,-178.682,5.654,148.602
C06182=1216.219,88.910,-47.798,-178.680,5.655,148.601
C06183=1216.215,89.159,-47.817,-178.678,5.655,148.600
C06184=1216.210,89.409,-47.835,-178.675,5.656,148.600
C06185=1216.205,89.658,-47.853,-178.673,5.657,148.599
C06186=1216.200,89.907,-47.871,-178.670,5.658,148.599
C06187=1216.195,90.156,-47.889,-178.667,5.659,148.598
C06188=1216.191,90.406,-47.907,-178.665,5.660,148.598
C06189=1216.185,90.656,-47.926,-178.662,5.660,148.597
C06190=1216.180,90.905,-47.944,-178.660,5.661,148.596
C06191=1216.175,91.154,-47.961,-178.657,5.663,148.596
C06192=1216.171,91.402,-47.980,-178.654,5.663,148.595
C06193=1216.167,91.652,-47.999,-178.652,5.664,148.595
C06194=1216.162,91.901,-48.017,-178.650,5.665,148.594
C06195=1216.157,92.151,-48.034,-178.646,5.666,148.594
C06196=1216.151,92.400,-48.053,-178.644,5.667,148.593
C06197=1216.147,92.650,-48.071,-178.642,5.668,148.593
C06198=1216.142,92.899,-48.090,-178.639,5.668,148.592
C06199=1216.137,93.148,-48.108,-178.637,5.669,148.591
C06200=1216.132,93.397,-48.126,-178.634,5.671,148.591
C06201=1216.127,93.646,-48.145,-178.631,5.671,148.590
C06202=1216.123,93.896,-48.164,-178.629,5.672,148.590
C06203=1216.118,94.145,-48.182,-178.626,5.673,148.589
C06204=1216.113,94.394,-48.200,-178.623,5.674,148.588
C06205=1216.108,94.644,-48.219,-178.621,5.675,148.588
C06206=1216.103,94.893,-48.237,-178.618,5.676,148.587
C06207=1216.098,95.142,-48.255,-178.616,5.677,148.587
C06208=1216.093,95.391,-48.273,-178.613,5.678,148.586
C06209=1216.089,95.641,-48.292,-178.611,5.679,148.586
C06210=1216.084,95.890,-48.311,-178.608,5.679,148.585
C06211=1216.079,96.139,-48.329,-178.606,5.680,148.585
C06212=1216.075,96.389,-48.347,-178.603,5.682,148.584
C06213=1216.069,96.638,-48.367,-178.600,5.682,148.584
C06214=1216.064,96.887,-48.384,-178.598,5.683,148.583
C06215=1216.059,97.136,-48.402,-178.596,5.684,148.582
C06216=1216.055,97.385,-48.422,-178.593,5.685,148.582
C06217=1216.050,97.635,-48.440,-178.590,5.686,148.581
C06218=1216.045,97.884,-48.458,-178.588,5.687,148.581
C06219=1216.041,98.133,-48.477,-178.585,5.688,148.580
C06220=1216.035,98.383,-48.496,-178.582,5.689,148.580
C06221=1216.031,98.631,-48.514,-178.580,5.690,148.579
C06222=1216.026,98.881,-48.533,-178.577,5.690,148.578
C06223=1216.021,99.131,-48.551,-178.575,5.691,148.578
C06224=1216.016,99.379,-48.570,-178.572,5.693,148.577
C06225=1216.012,99.629,-48.588,-178.569,5.693,148.577
C06226=1216.006,99.878,-48.608,-178.567,5.694,148.576
C06227=1216.001,100.127,-48.626,-178.565,5.695,148.576
C06228=1215.997,100.377,-48.645,-178.562,5.697,148.575
C06229=1215.992,100.626,-48.663,-178.559,5.697,148.575
C06230=1215.988,100.875,-48.682,-178.557,5.698,148.574
C06231=1215.982,101.125,-48.701,-178.555,5.699,148.574
C06232=1215.977,101.373,-48.720,-178.551,5.700,148.573
C06233=1215.972,101.623,-48.739,-178.549,5.701,148.573
C06234=1215.968,101.872,-48.757,-178.547,5.702,148.572
C06235=1215.963,102.121,-48.775,-178.543,5.703,148.571
C06236=1215.958,102.371,-48.795,-178.541,5.704,148.571
C06237=1215.953,102.620,-48.813,-178.539,5.705,148.570
C06238=1215.948,102.869,-48.833,-178.537,5.706,148.570
C06239=1215.944,103.119,-48.851,-178.533,5.707,148.569
C06240=1215.938,103.368,-48.870,-178.531,5.708,148.568
C06241=1215.934,103.617,-48.889,-178.529,5.709,148.568
C06242=1215.929,103.866,-48.907,-178.526,5.709,148.567
C06243=1215.925,104.116,-48.926,-178.523,5.711,148.567
C06244=1215.920,104.365,-48.944,-178.521,5.712,148.566
C06245=1215.915,104.614,-48.964,-178.518,5.712,148.566
C06246=1215.910,104.863,-48.983,-178.515,5.714,148.565
C06247=1215.905,105.112,-49.001,-178.513,5.715,148.565
C06248=1215.901,105.362,-49.020,-178.511,5.716,148.564
C06249=1215.895,105.610,-49.040,-178.507,5.717,148.564
C06250=1215.891,105.860,-49.058,-178.505,5.718,148.563
C06251=1215.886,106.109,-49.077,-178.503,5.719,148.563
C06252=1215.881,106.359,-49.097,-178.500,5.719,148.562
C06253=1215.876,106.608,-49.115,-178.497,5.721,148.562
C06254=1215.871,106.858,-49.135,-178.495,5.722,148.561
C06255=1215.866,107.125,-49.155,-178.492,5.722,148.560
C06256=1215.861,107.394,-49.175,-178.489,5.724,148.560
C06257=1215.856,107.662,-49.196,-178.487,5.725,148.559
C06258=1215.850,107.930,-49.217,-178.484,5.726,148.559
C06259=1215.846,108.180,-49.235,-178.482,5.727,148.558
C06260=1215.841,108.429,-49.254,-178.478,5.728,148.557
C06261=1215.837,108.678,-49.273,-178.476,5.729,148.557
C06262=1215.831,108.927,-49.293,-178.474,5.730,148.556
C06263=1215.826,109.177,-49.312,-178.470,5.731,148.556
C06264=1215.822,109.426,-49.330,-178.468,5.732,148.555
C06265=1215.817,109.675,-49.350,-178.466,5.733,148.555
C06266=1215.812,109.924,-49.369,-178.464,5.734,148.554
C06267=1215.807,110.174,-49.388,-178.460,5.735,148.554
C06268=1215.802,110.422,-49.408,-178.458,5.736,148.553
C06269=1215.798,110.672,-49.426,-178.456,5.737,148.553
C06270=1215.793,110.922,-49.446,-178.453,5.738,148.552
C06271=1215.788,111.171,-49.465,-178.450,5.739,148.552
C06272=1215.784,111.420,-49.484,-178.448,5.740,148.551
C06273=1215.778,111.669,-49.503,-178.445,5.742,148.551
C06274=1215.774,111.918,-49.523,-178.442,5.742,148.550
C06275=1215.769,112.167,-49.542,-178.440,5.743,148.550
C06276=1215.764,112.417,-49.561,-178.437,5.745,148.549
C06277=1215.759,112.665,-49.580,-178.435,5.746,148.548
C06278=1215.755,112.915,-49.599,-178.432,5.746,148.548
C06279=1215.750,113.165,-49.618,-178.429,5.748,148.547
C06280=1215.745,113.414,-49.638,-178.427,5.749,148.547
C06281=1215.740,113.663,-49.657,-178.425,5.749,148.546
C06282=1215.735,113.912,-49.676,-178.422,5.751,148.546
C06283=1215.730,114.161,-49.696,-178.419,5.752,148.545
C06284=1215.725,114.410,-49.715,-178.417,5.752,148.545
C06285=1215.720,114.660,-49.735,-178.414,5.754,148.544
C06286=1215.716,114.909,-49.754,-178.412,5.755,148.544
C06287=1215.711,115.158,-49.773,-178.409,5.756,148.543
C06288=1215.706,115.408,-49.793,-178.406,5.757,148.543
C06289=1215.701,115.656,-49.812,-178.404,5.758,148.542
C06290=1215.697,115.906,-49.831,-178.401,5.760,148.542
C06291=1215.692,116.155,-49.851,-178.399,5.760,148.541
C06292=1215.687,116.404,-49.871,-178.396,5.761,148.541
C06293=1215.682,116.653,-49.890,-178.393,5.763,148.540
C06294=1215.678,116.903,-49.910,-178.391,5.764,148.540
C06295=1215.673,117.151,-49.929,-178.389,5.764,148.539
C06296=1215.668,117.401,-49.948,-178.385,5.766,148.538
C06297=1215.663,117.650,-49.968,-178.383,5.767,148.538
C06298=1215.658,117.899,-49.987,-178.381,5.767,148.537
C06299=1215.654,118.149,-50.007,-178.378,5.769,148.537
C06300=1215.649,118.397,-50.026,-178.375,5.770,148.536
C06301=1215.644,118.646,-50.046,-178.373,5.771,148.536
C06302=1215.640,118.896,-50.066,-178.370,5.772,148.535
C06303=1215.634,119.145,-50.085,-178.368,5.773,148.535
C06304=1215.630,119.394,-50.105,-178.365,5.774,148.534
C06305=1215.625,119.644,-50.124,-178.363,5.775,148.534
C06306=1215.620,119.893,-50.144,-178.360,5.776,148.533
C06307=1215.615,120.142,-50.164,-178.357,5.778,148.533
C06308=1215.611,120.391,-50.183,-178.355,5.778,148.532
C06309=1215.606,120.640,-50.202,-178.352,5.780,148.532
C06310=1215.601,120.889,-50.222,-178.349,5.781,148.531
C06311=1215.597,121.138,-50.242,-178.347,5.782,148.531
C06312=1215.592,121.388,-50.262,-178.344,5.783,148.530
C06313=1215.586,121.637,-50.281,-178.342,5.784,148.530
C06314=1215.582,121.886,-50.301,-178.339,5.786,148.529
C06315=1215.577,122.135,-50.321,-178.337,5.787,148.529
C06316=1215.572,122.384,-50.341,-178.334,5.787,148.528
C06317=1215.567,122.634,-50.360,-178.331,5.789,148.527
C06318=1215.563,122.883,-50.381,-178.329,5.790,148.527
C06319=1215.558,123.132,-50.400,-178.326,5.791,148.526
C06320=1215.553,123.381,-50.420,-178.324,5.792,148.526
C06321=1215.548,123.630,-50.440,-178.321,5.793,148.525
C06322=1215.544,123.880,-50.460,-178.318,5.794,148.525
C06323=1215.539,124.129,-50.479,-178.316,5.795,148.524
C06324=1215.534,124.377,-50.499,-178.313,5.797,148.524
C06325=1215.529,124.627,-50.519,-178.311,5.798,148.523
C06326=1215.524,124.877,-50.539,-178.309,5.799,148.523
C06327=1215.520,125.126,-50.559,-178.306,5.800,148.522
C06328=1215.514,125.374,-50.578,-178.303,5.801,148.522
C06329=1215.510,125.623,-50.599,-178.300,5.802,148.521
C06330=1215.505,125.873,-50.618,-178.298,5.803,148.521
C06331=1215.501,126.122,-50.639,-178.296,5.804,148.520
C06332=1215.496,126.371,-50.658,-178.293,5.806,148.520
C06333=1215.491,126.620,-50.678,-178.290,5.806,148.519
C06334=1215.486,126.869,-50.698,-178.288,5.808,148.519
C06335=1215.482,127.119,-50.718,-178.285,5.809,148.518
C06336=1215.477,127.368,-50.738,-178.282,5.811,148.518
C06337=1215.472,127.617,-50.758,-178.280,5.811,148.517
C06338=1215.467,127.866,-50.778,-178.278,5.812,148.517
C06339=1215.463,128.115,-50.797,-178.274,5.814,148.516
C06340=1215.458,128.364,-50.818,-178.272,5.815,148.516
C06341=1215.453,128.614,-50.837,-178.270,5.816,148.515
C06342=1215.448,128.863,-50.858,-178.267,5.817,148.515
C06343=1215.444,129.112,-50.879,-178.264,5.819,148.514
C06344=1215.438,129.361,-50.898,-178.262,5.819,148.514
C06345=1215.434,129.610,-50.918,-178.260,5.820,148.513
C06346=1215.429,129.859,-50.938,-178.256,5.822,148.513
C06347=1215.425,130.108,-50.958,-178.254,5.823,148.512
C06348=1215.420,130.358,-50.978,-178.251,5.824,148.512
C06349=1215.415,130.607,-50.999,-178.249,5.825,148.511
C06350=1215.411,130.856,-51.019,-178.246,5.827,148.511
C06351=1215.405,131.105,-51.039,-178.244,5.828,148.510
C06352=1215.401,131.354,-51.059,-178.241,5.829,148.510
C06353=1215.396,131.603,-51.079,-178.238,5.830,148.509
C06354=1215.391,131.853,-51.100,-178.236,5.831,148.509
C06355=1215.386,132.102,-51.120,-178.233,5.832,148.508
C06356=1215.382,132.351,-51.140,-178.231,5.833,148.508
C06357=1215.377,132.600,-51.160,-178.228,5.835,148.507
C06358=1215.373,132.849,-51.180,-178.226,5.836,148.507
C06359=1215.367,133.118,-51.202,-178.223,5.837,148.506
C06360=1215.362,133.386,-51.225,-178.220,5.839,148.506
C06361=1215.357,133.655,-51.246,-178.217,5.840,148.505
C06362=1215.352,133.923,-51.268,-178.214,5.841,148.505
C06363=1215.347,134.172,-51.288,-178.212,5.842,148.504
C06364=1215.342,134.422,-51.308,-178.209,5.844,148.504
C06365=1215.337,134.671,-51.329,-178.207,5.845,148.503
C06366=1215.333,134.920,-51.349,-178.204,5.846,148.503
C06367=1215.328,135.169,-51.370,-178.201,5.847,148.502
C06368=1215.323,135.418,-51.391,-178.199,5.849,148.502
C06369=1215.318,135.668,-51.410,-178.197,5.850,148.501
C06370=1215.314,135.917,-51.431,-178.194,5.851,148.501
C06371=1215.309,136.166,-51.451,-178.191,5.852,148.500
C06372=1215.304,136.415,-51.472,-178.188,5.854,148.500
C06373=1215.300,136.664,-51.492,-178.186,5.855,148.499
C06374=1215.295,136.913,-51.513,-178.183,5.856,148.499
C06375=1215.290,137.163,-51.533,-178.181,5.857,148.498
C06376=1215.285,137.411,-51.553,-178.179,5.858,148.498
C06377=1215.280,137.660,-51.573,-178.176,5.859,148.497
C06378=1215.275,137.909,-51.594,-178.173,5.860,148.497
C06379=1215.271,138.158,-51.615,-178.170,5.862,148.496
C06380=1215.266,138.407,-51.636,-178.168,5.863,148.496
C06381=1215.261,138.656,-51.656,-178.166,5.865,148.495
C06382=1215.257,138.905,-51.677,-178.163,5.865,148.495
C06383=1215.252,139.155,-51.697,-178.160,5.867,148.494
C06384=1215.247,139.404,-51.718,-178.158,5.868,148.494
C06385=1215.243,139.652,-51.738,-178.155,5.869,148.493
C06386=1215.238,139.902,-51.759,-178.153,5.870,148.493
C06387=1215.233,140.151,-51.780,-178.150,5.872,148.492
C06388=1215.229,140.401,-51.801,-178.148,5.873,148.492
C06389=1215.224,140.650,-51.821,-178.144,5.874,148.491
C06390=1215.219,140.899,-51.842,-178.142,5.875,148.491
C06391=1215.215,141.148,-51.863,-178.140,5.877,148.491
C06392=1215.210,141.397,-51.883,-178.137,5.878,148.490
C06393=1215.205,141.646,-51.904,-178.134,5.879,148.490
C06394=1215.200,141.895,-51.924,-178.132,5.880,148.489
C06395=1215.195,142.144,-51.945,-178.129,5.882,148.489
C06396=1215.191,142.393,-51.966,-178.126,5.884,148.488
C06397=1215.186,142.642,-51.987,-178.124,5.884,148.488
C06398=1215.181,142.891,-52.007,-178.121,5.886,148.487
C06399=1215.176,143.141,-52.028,-178.119,5.887,148.487
C06400=1215.172,143.390,-52.048,-178.116,5.889,148.486
C06401=1215.166,143.639,-52.069,-178.114,5.890,148.486
C06402=1215.162,143.888,-52.090,-178.111,5.891,148.485
C06403=1215.157,144.136,-52.111,-178.108,5.892,148.485
C06404=1215.153,144.386,-52.132,-178.106,5.894,148.484
C06405=1215.148,144.635,-52.153,-178.103,5.894,148.484
C06406=1215.144,144.884,-52.173,-178.101,5.896,148.483
C06407=1215.139,145.134,-52.194,-178.098,5.897,148.483
C06408=1215.134,145.383,-52.215,-178.095,5.899,148.482
C06409=1215.129,145.631,-52.236,-178.093,5.900,148.482
C06410=1215.124,145.880,-52.257,-178.090,5.901,148.482
C06411=1215.120,146.129,-52.278,-178.088,5.902,148.481
C06412=1215.114,146.379,-52.299,-178.085,5.904,148.481
C06413=1215.111,146.628,-52.320,-178.083,5.906,148.480
C06414=1215.106,146.877,-52.341,-178.080,5.906,148.480
C06415=1215.101,147.126,-52.362,-178.077,5.908,148.479
C06416=1215.096,147.375,-52.383,-178.075,5.909,148.479
C06417=1215.091,147.624,-52.404,-178.072,5.911,148.478
C06418=1215.087,147.873,-52.425,-178.070,5.911,148.478
C06419=1215.082,148.122,-52.446,-178.067,5.913,148.477
C06420=1215.077,148.371,-52.468,-178.065,5.914,148.477
C06421=1215.073,148.620,-52.488,-178.062,5.916,148.477
C06422=1215.068,148.870,-52.509,-178.059,5.916,148.476
C06423=1215.063,149.119,-52.530,-178.057,5.918,148.476
C06424=1215.058,149.367,-52.551,-178.054,5.920,148.475
C06425=1215.054,149.617,-52.572,-178.051,5.921,148.475
C06426=1215.049,149.866,-52.594,-178.049,5.922,148.474
C06427=1215.045,150.115,-52.614,-178.047,5.923,148.474
C06428=1215.039,150.364,-52.635,-178.043,5.925,148.473
C06429=1215.035,150.613,-52.657,-178.041,5.926,148.473
C06430=1215.030,150.862,-52.677,-178.039,5.928,148.472
C06431=1215.026,151.111,-52.699,-178.036,5.929,148.472
C06432=1215.021,151.360,-52.720,-178.033,5.930,148.471
C06433=1215.015,151.609,-52.741,-178.031,5.932,148.471
C06434=1215.011,151.858,-52.762,-178.028,5.932,148.470
C06435=1215.007,152.108,-52.784,-178.026,5.934,148.470
C06436=1215.002,152.356,-52.805,-178.023,5.935,148.470
C06437=1214.997,152.606,-52.826,-178.021,5.937,148.469
C06438=1214.993,152.854,-52.848,-178.018,5.939,148.469
C06439=1214.987,153.103,-52.869,-178.015,5.940,148.468
C06440=1214.983,153.352,-52.891,-178.013,5.941,148.468
C06441=1214.978,153.602,-52.912,-178.010,5.942,148.467
C06442=1214.974,153.850,-52.933,-178.008,5.944,148.467
C06443=1214.969,154.099,-52.954,-178.005,5.945,148.466
C06444=1214.964,154.349,-52.976,-178.002,5.946,148.466
C06445=1214.959,154.598,-52.997,-178.000,5.948,148.466
C06446=1214.954,154.847,-53.018,-177.998,5.949,148.465
C06447=1214.951,155.096,-53.040,-177.994,5.950,148.465
C06448=1214.946,155.345,-53.061,-177.992,5.951,148.464
C06449=1214.941,155.594,-53.082,-177.990,5.953,148.464
C06450=1214.936,155.843,-53.103,-177.987,5.955,148.463
C06451=1214.931,156.092,-53.125,-177.984,5.956,148.463
C06452=1214.926,156.341,-53.147,-177.982,5.958,148.462
C06453=1214.921,156.590,-53.168,-177.980,5.958,148.462
C06454=1214.918,156.839,-53.189,-177.976,5.960,148.461
C06455=1214.913,157.088,-53.211,-177.974,5.962,148.461
C06456=1214.908,157.337,-53.232,-177.972,5.963,148.461
C06457=1214.903,157.586,-53.254,-177.968,5.964,148.460
C06458=1214.899,157.835,-53.276,-177.966,5.965,148.460
C06459=1214.893,158.084,-53.297,-177.964,5.967,148.459
C06460=1214.889,158.334,-53.319,-177.961,5.969,148.459
C06461=1214.884,158.582,-53.341,-177.958,5.969,148.458
C06462=1214.879,158.831,-53.362,-177.956,5.971,148.458
C06463=1214.875,159.100,-53.385,-177.953,5.973,148.458
C06464=1214.869,159.369,-53.408,-177.950,5.975,148.457
C06465=1214.864,159.638,-53.431,-177.948,5.976,148.457
C06466=1214.859,159.907,-53.455,-177.945,5.977,148.456
C06467=1214.855,160.157,-53.477,-177.942,5.979,148.456
C06468=1214.850,160.406,-53.498,-177.939,5.981,148.455
C06469=1214.845,160.654,-53.520,-177.937,5.981,148.455
C06470=1214.841,160.904,-53.542,-177.934,5.983,148.454
C06471=1214.836,161.152,-53.564,-177.932,5.984,148.454
C06472=1214.832,161.402,-53.586,-177.929,5.986,148.454
C06473=1214.826,161.651,-53.607,-177.926,5.987,148.453
C06474=1214.821,161.899,-53.628,-177.924,5.988,148.453
C06475=1214.817,162.149,-53.650,-177.921,5.990,148.452
C06476=1214.812,162.397,-53.672,-177.919,5.992,148.452
C06477=1214.808,162.647,-53.694,-177.916,5.993,148.451
C06478=1214.803,162.895,-53.716,-177.914,5.994,148.451
C06479=1214.798,163.144,-53.737,-177.911,5.996,148.450
C06480=1214.794,163.393,-53.760,-177.909,5.997,148.450
C06481=1214.789,163.643,-53.780,-177.906,5.999,148.449
C06482=1214.785,163.892,-53.803,-177.903,6.000,148.449
C06483=1214.780,164.141,-53.824,-177.901,6.001,148.449
C06484=1214.776,164.390,-53.846,-177.898,6.003,148.448
C06485=1214.771,164.639,-53.868,-177.896,6.004,148.448
C06486=1214.766,164.887,-53.890,-177.893,6.006,148.447
C06487=1214.761,165.137,-53.912,-177.890,6.008,148.447
C06488=1214.756,165.386,-53.934,-177.888,6.009,148.447
C06489=1214.752,165.635,-53.956,-177.885,6.010,148.446
C06490=1214.747,165.884,-53.978,-177.882,6.012,148.446
C06491=1214.742,166.133,-54.000,-177.880,6.013,148.445
C06492=1214.738,166.382,-54.021,-177.878,6.015,148.445
C06493=1214.733,166.631,-54.043,-177.874,6.016,148.444
C06494=1214.728,166.880,-54.065,-177.872,6.017,148.444
C06495=1214.724,167.129,-54.087,-177.870,6.019,148.444
C06496=1214.719,167.377,-54.110,-177.867,6.021,148.443
C06497=1214.715,167.627,-54.132,-177.865,6.022,148.443
C06498=1214.710,167.875,-54.154,-177.862,6.023,148.442
C06499=1214.706,168.125,-54.176,-177.859,6.025,148.442
C06500=1214.701,168.373,-54.198,-177.856,6.027,148.441
C06501=1214.696,168.622,-54.220,-177.854,6.028,148.441
C06502=1214.691,168.871,-54.242,-177.851,6.029,148.441
C06503=1214.686,169.121,-54.264,-177.849,6.031,148.440
C06504=1214.682,169.369,-54.286,-177.846,6.032,148.440
C06505=1214.678,169.618,-54.308,-177.844,6.034,148.439
C06506=1214.672,169.867,-54.331,-177.841,6.036,148.439
C06507=1214.668,170.116,-54.353,-177.839,6.036,148.438
C06508=1214.663,170.365,-54.374,-177.836,6.038,148.438
C06509=1214.659,170.614,-54.397,-177.833,6.040,148.438
C06510=1214.653,170.863,-54.420,-177.831,6.041,148.437
C06511=1214.649,171.112,-54.442,-177.828,6.043,148.437
C06512=1214.645,171.361,-54.464,-177.825,6.044,148.436
C06513=1214.640,171.610,-54.485,-177.823,6.046,148.436
C06514=1214.635,171.859,-54.509,-177.821,6.047,148.436
C06515=1214.630,172.108,-54.530,-177.818,6.049,148.435
C06516=1214.626,172.357,-54.552,-177.815,6.051,148.435
C06517=1214.621,172.606,-54.575,-177.813,6.051,148.434
C06518=1214.617,172.855,-54.597,-177.810,6.053,148.434
C06519=1214.612,173.104,-54.619,-177.807,6.055,148.434
C06520=1214.607,173.353,-54.642,-177.805,6.056,148.433
C06521=1214.603,173.602,-54.665,-177.803,6.058,148.433
C06522=1214.598,173.850,-54.686,-177.799,6.059,148.432
C06523=1214.593,174.100,-54.709,-177.797,6.061,148.432
C06524=1214.589,174.349,-54.732,-177.795,6.062,148.431
C06525=1214.584,174.597,-54.753,-177.792,6.064,148.431
C06526=1214.579,174.846,-54.777,-177.789,6.066,148.431
C06527=1214.574,175.095,-54.798,-177.787,6.066,148.430
C06528=1214.570,175.344,-54.820,-177.784,6.068,148.430
C06529=1214.565,175.593,-54.844,-177.781,6.070,148.429
C06530=1214.561,175.842,-54.865,-177.779,6.072,148.429
C06531=1214.556,176.091,-54.889,-177.777,6.073,148.429
C06532=1214.552,176.340,-54.911,-177.774,6.075,148.428
C06533=1214.547,176.588,-54.933,-177.771,6.076,148.428
C06534=1214.542,176.838,-54.956,-177.768,6.078,148.427
C06535=1214.538,177.087,-54.978,-177.766,6.079,148.427
C06536=1214.532,177.336,-55.001,-177.763,6.081,148.427
C06537=1214.528,177.585,-55.023,-177.761,6.083,148.426
C06538=1214.524,177.834,-55.046,-177.758,6.084,148.426
C06539=1214.519,178.083,-55.068,-177.756,6.085,148.425
C06540=1214.515,178.332,-55.091,-177.753,6.087,148.425
C06541=1214.510,178.581,-55.114,-177.750,6.089,148.425
C06542=1214.505,178.829,-55.136,-177.748,6.091,148.424
C06543=1214.500,179.078,-55.159,-177.746,6.092,148.424
C06544=1214.496,179.328,-55.181,-177.743,6.093,148.424
C06545=1214.491,179.576,-55.204,-177.740,6.095,148.423
C06546=1214.487,179.825,-55.226,-177.737,6.097,148.423
C06547=1214.482,180.074,-55.250,-177.735,6.098,148.422
C06548=1214.478,180.323,-55.272,-177.732,6.099,148.422
C06549=1214.472,180.572,-55.295,-177.730,6.101,148.421
C06550=1214.468,180.821,-55.317,-177.727,6.103,148.421
C06551=1214.464,181.070,-55.341,-177.725,6.104,148.421
C06552=1214.459,181.319,-55.363,-177.722,6.106,148.420
C06553=1214.454,181.567,-55.386,-177.719,6.107,148.420
C06554=1214.449,181.816,-55.409,-177.716,6.109,148.419
C06555=1214.445,182.066,-55.431,-177.714,6.110,148.419
C06556=1214.440,182.315,-55.455,-177.712,6.112,148.419
C06557=1214.436,182.563,-55.477,-177.709,6.114,148.418
C06558=1214.431,182.812,-55.500,-177.706,6.116,148.418
C06559=1214.426,183.062,-55.523,-177.704,6.117,148.418
C06560=1214.422,183.310,-55.546,-177.701,6.118,148.417
C06561=1214.417,183.559,-55.569,-177.699,6.120,148.417
C06562=1214.413,183.808,-55.591,-177.696,6.122,148.416
C06563=1214.408,184.057,-55.614,-177.693,6.124,148.416
C06564=1214.403,184.306,-55.638,-177.691,6.125,148.416
C06565=1214.399,184.555,-55.660,-177.688,6.126,148.415
C06566=1214.394,184.804,-55.683,-177.686,6.128,148.415
C06567=1214.389,185.073,-55.708,-177.683,6.130,148.414
C06568=1214.384,185.342,-55.733,-177.680,6.132,148.414
C06569=1214.379,185.612,-55.758,-177.677,6.133,148.414
C06570=1214.374,185.881,-55.782,-177.675,6.135,148.413
C06571=1214.369,186.130,-55.806,-177.672,6.137,148.413
C06572=1214.365,186.380,-55.829,-177.669,6.139,148.412
C06573=1214.360,186.629,-55.852,-177.667,6.140,148.412
C06574=1214.356,186.878,-55.874,-177.664,6.141,148.412
C06575=1214.351,187.127,-55.898,-177.662,6.143,148.411
C06576=1214.346,187.375,-55.921,-177.659,6.145,148.411
C06577=1214.342,187.624,-55.943,-177.656,6.147,148.411
C06578=1214.337,187.873,-55.967,-177.654,6.148,148.410
C06579=1214.332,188.122,-55.990,-177.651,6.150,148.410
C06580=1214.328,188.371,-56.014,-177.649,6.152,148.409
C06581=1214.324,188.620,-56.036,-177.646,6.153,148.409
C06582=1214.319,188.869,-56.060,-177.643,6.155,148.409
C06583=1214.314,189.117,-56.083,-177.640,6.157,148.408
C06584=1214.309,189.366,-56.106,-177.638,6.158,148.408
C06585=1214.305,189.615,-56.129,-177.636,6.160,148.407
C06586=1214.300,189.864,-56.152,-177.633,6.161,148.407
C06587=1214.296,190.113,-56.175,-177.630,6.163,148.407
C06588=1214.291,190.362,-56.199,-177.628,6.165,148.406
C06589=1214.286,190.611,-56.222,-177.626,6.166,148.406
C06590=1214.282,190.860,-56.246,-177.623,6.168,148.406
C06591=1214.278,191.109,-56.268,-177.620,6.170,148.405
C06592=1214.272,191.357,-56.291,-177.618,6.172,148.405
C06593=1214.268,191.606,-56.315,-177.615,6.173,148.405
C06594=1214.263,191.855,-56.338,-177.612,6.175,148.404
C06595=1214.258,192.104,-56.361,-177.610,6.176,148.404
C06596=1214.254,192.353,-56.385,-177.607,6.178,148.403
C06597=1214.249,192.602,-56.409,-177.604,6.179,148.403
C06598=1214.245,192.850,-56.432,-177.602,6.181,148.403
C06599=1214.240,193.099,-56.455,-177.599,6.183,148.402
C06600=1214.236,193.348,-56.478,-177.597,6.185,148.402
C06601=1214.231,193.598,-56.502,-177.594,6.187,148.402
C06602=1214.226,193.847,-56.525,-177.592,6.188,148.401
C06603=1214.222,194.095,-56.549,-177.589,6.190,148.401
C06604=1214.217,194.344,-56.572,-177.587,6.191,148.401
C06605=1214.213,194.593,-56.596,-177.584,6.193,148.400
C06606=1214.208,194.842,-56.619,-177.581,6.195,148.400
C06607=1214.203,195.090,-56.643,-177.579,6.197,148.400
C06608=1214.199,195.339,-56.667,-177.576,6.198,148.399
C06609=1214.194,195.589,-56.690,-177.574,6.200,148.399
C06610=1214.189,195.838,-56.713,-177.571,6.202,148.398
C06611=1214.185,196.086,-56.737,-177.569,6.203,148.398
C06612=1214.181,196.335,-56.760,-177.565,6.205,148.398
C06613=1214.176,196.584,-56.784,-177.563,6.207,148.397
C06614=1214.172,196.832,-56.808,-177.560,6.209,148.397
C06615=1214.167,197.081,-56.831,-177.557,6.210,148.397
C06616=1214.163,197.330,-56.854,-177.555,6.211,148.396
C06617=1214.157,197.579,-56.879,-177.553,6.213,148.396
C06618=1214.153,197.828,-56.902,-177.550,6.215,148.395
C06619=1214.148,198.077,-56.926,-177.547,6.217,148.395
C06620=1214.144,198.325,-56.950,-177.545,6.219,148.395
C06621=1214.139,198.574,-56.973,-177.542,6.221,148.394
C06622=1214.134,198.823,-56.997,-177.540,6.222,148.394
C06623=1214.130,199.072,-57.021,-177.537,6.224,148.394
C06624=1214.125,199.321,-57.044,-177.535,6.225,148.393
C06625=1214.121,199.569,-57.068,-177.532,6.227,148.393
C06626=1214.116,199.818,-57.091,-177.529,6.229,148.393
C06627=1214.112,200.067,-57.115,-177.527,6.231,148.392
C06628=1214.107,200.316,-57.139,-177.524,6.233,148.392
C06629=1214.103,200.564,-57.163,-177.522,6.234,148.392
C06630=1214.098,200.813,-57.186,-177.519,6.236,148.391
C06631=1214.094,201.062,-57.211,-177.516,6.238,148.391
C06632=1214.089,201.312,-57.235,-177.514,6.240,148.391
C06633=1214.084,201.560,-57.259,-177.512,6.241,148.390
C06634=1214.080,201.809,-57.282,-177.509,6.243,148.390
C06635=1214.075,202.058,-57.306,-177.506,6.245,148.390
C06636=1214.070,202.307,-57.330,-177.504,6.247,148.389
C06637=1214.066,202.555,-57.354,-177.501,6.248,148.389
C06638=1214.061,202.804,-57.377,-177.498,6.250,148.389
C06639=1214.056,203.053,-57.402,-177.496,6.252,148.388
C06640=1214.052,203.302,-57.425,-177.493,6.254,148.388
C06641=1214.048,203.551,-57.449,-177.490,6.256,148.388
C06642=1214.043,203.799,-57.473,-177.488,6.258,148.387
C06643=1214.039,204.048,-57.497,-177.485,6.259,148.387
C06644=1214.033,204.297,-57.522,-177.483,6.260,148.386
C06645=1214.029,204.545,-57.546,-177.480,6.262,148.386
C06646=1214.024,204.795,-57.569,-177.478,6.264,148.386
C06647=1214.021,205.044,-57.593,-177.475,6.266,148.385
C06648=1214.016,205.292,-57.617,-177.472,6.268,148.385
C06649=1214.011,205.541,-57.641,-177.470,6.270,148.385
C06650=1214.006,205.790,-57.665,-177.467,6.271,148.384
C06651=1214.002,206.038,-57.690,-177.465,6.273,148.384
C06652=1213.997,206.287,-57.713,-177.462,6.275,148.384
C06653=1213.993,206.537,-57.738,-177.459,6.277,148.383
C06654=1213.988,206.785,-57.762,-177.457,6.279,148.383
C06655=1213.984,207.033,-57.786,-177.454,6.281,148.383
C06656=1213.979,207.283,-57.810,-177.451,6.282,148.382
C06657=1213.974,207.531,-57.834,-177.449,6.283,148.382
C06658=1213.970,207.780,-57.859,-177.447,6.285,148.382
C06659=1213.965,208.029,-57.883,-177.444,6.287,148.381
C06660=1213.961,208.277,-57.907,-177.441,6.289,148.381
C06661=1213.956,208.527,-57.931,-177.439,6.291,148.381
C06662=1213.952,208.776,-57.956,-177.436,6.293,148.380
C06663=1213.947,209.024,-57.980,-177.433,6.294,148.380
C06664=1213.943,209.273,-58.004,-177.431,6.296,148.380
C06665=1213.938,209.521,-58.029,-177.429,6.298,148.380
C06666=1213.933,209.770,-58.053,-177.426,6.300,148.379
C06667=1213.929,210.019,-58.077,-177.423,6.302,148.379
C06668=1213.924,210.268,-58.102,-177.421,6.304,148.379
C06669=1213.920,210.517,-58.125,-177.418,6.306,148.378
C06670=1213.915,210.766,-58.150,-177.415,6.308,148.378
C06671=1213.911,211.036,-58.176,-177.413,6.310,148.378
C06672=1213.906,211.306,-58.203,-177.410,6.311,148.377
C06673=1213.900,211.576,-58.230,-177.406,6.314,148.377
C06674=1213.895,211.847,-58.256,-177.404,6.316,148.376
C06675=1213.891,212.096,-58.280,-177.401,6.317,148.376
C06676=1213.886,212.345,-58.305,-177.399,6.319,148.376
C06677=1213.882,212.593,-58.329,-177.396,6.321,148.376
C06678=1213.877,212.843,-58.354,-177.394,6.323,148.375
C06679=1213.873,213.091,-58.378,-177.391,6.325,148.375
C06680=1213.868,213.340,-58.403,-177.388,6.327,148.375
C06681=1213.863,213.588,-58.427,-177.386,6.329,148.374
C06682=1213.859,213.837,-58.452,-177.383,6.331,148.374
C06683=1213.855,214.086,-58.477,-177.381,6.332,148.374
C06684=1213.849,214.334,-58.501,-177.378,6.334,148.373
C06685=1213.846,214.583,-58.526,-177.375,6.336,148.373
C06686=1213.840,214.832,-58.550,-177.373,6.337,148.373
C06687=1213.836,215.081,-58.574,-177.371,6.339,148.372
C06688=1213.832,215.330,-58.599,-177.368,6.341,148.372
C06689=1213.827,215.578,-58.623,-177.365,6.343,148.372
C06690=1213.822,215.827,-58.648,-177.363,6.345,148.371
C06691=1213.819,216.076,-58.673,-177.360,6.347,148.371
C06692=1213.813,216.324,-58.698,-177.358,6.349,148.371
C06693=1213.810,216.574,-58.722,-177.355,6.350,148.370
C06694=1213.804,216.822,-58.747,-177.353,6.352,148.370
C06695=1213.799,217.071,-58.772,-177.350,6.354,148.370
C06696=1213.796,217.320,-58.796,-177.347,6.356,148.369
C06697=1213.791,217.568,-58.822,-177.345,6.358,148.369
C06698=1213.787,217.817,-58.846,-177.342,6.360,148.369
C06699=1213.782,218.066,-58.871,-177.339,6.361,148.368
C06700=1213.777,218.315,-58.895,-177.337,6.363,148.368
C06701=1213.773,218.563,-58.921,-177.335,6.365,148.368
C06702=1213.768,218.812,-58.945,-177.332,6.367,148.368
C06703=1213.764,219.061,-58.970,-177.329,6.369,148.367
C06704=1213.759,219.309,-58.995,-177.327,6.371,148.367
C06705=1213.754,219.558,-59.020,-177.323,6.374,148.367
C06706=1213.751,219.807,-59.044,-177.321,6.376,148.366
C06707=1213.746,220.055,-59.069,-177.318,6.377,148.366
C06708=1213.741,220.305,-59.095,-177.316,6.379,148.366
C06709=1213.737,220.553,-59.119,-177.313,6.381,148.365
C06710=1213.733,220.802,-59.144,-177.311,6.383,148.365
C06711=1213.727,221.050,-59.169,-177.308,6.385,148.365
C06712=1213.723,221.300,-59.194,-177.306,6.387,148.365
C06713=1213.719,221.548,-59.219,-177.303,6.389,148.364
C06714=1213.714,221.796,-59.244,-177.300,6.391,148.364
C06715=1213.709,222.045,-59.269,-177.298,6.393,148.364
C06716=1213.705,222.294,-59.293,-177.295,6.394,148.363
C06717=1213.701,222.543,-59.318,-177.293,6.397,148.363
C06718=1213.696,222.791,-59.344,-177.290,6.398,148.363
C06719=1213.691,223.041,-59.369,-177.288,6.400,148.363
C06720=1213.687,223.288,-59.394,-177.285,6.402,148.362
C06721=1213.683,223.538,-59.419,-177.282,6.404,148.362
C06722=1213.678,223.786,-59.444,-177.280,6.406,148.362
C06723=1213.673,224.035,-59.469,-177.277,6.408,148.361
C06724=1213.668,224.283,-59.494,-177.275,6.410,148.361
C06725=1213.665,224.533,-59.519,-177.272,6.412,148.361
C06726=1213.660,224.781,-59.544,-177.270,6.413,148.360
C06727=1213.656,225.029,-59.570,-177.267,6.415,148.360
C06728=1213.650,225.278,-59.595,-177.264,6.417,148.360
C06729=1213.646,225.527,-59.620,-177.262,6.419,148.360
C06730=1213.641,225.776,-59.645,-177.260,6.421,148.359
C06731=1213.638,226.024,-59.670,-177.257,6.423,148.359
C06732=1213.633,226.274,-59.695,-177.254,6.425,148.359
C06733=1213.628,226.522,-59.721,-177.252,6.427,148.358
C06734=1213.624,226.771,-59.746,-177.249,6.429,148.358
C06735=1213.619,227.019,-59.771,-177.246,6.430,148.358
C06736=1213.615,227.268,-59.797,-177.244,6.433,148.358
C06737=1213.610,227.516,-59.822,-177.242,6.434,148.357
C06738=1213.605,227.766,-59.847,-177.239,6.436,148.357
C06739=1213.601,228.014,-59.873,-177.236,6.438,148.357
C06740=1213.597,228.262,-59.898,-177.233,6.441,148.356
C06741=1213.592,228.512,-59.923,-177.231,6.443,148.356
C06742=1213.588,228.760,-59.948,-177.228,6.445,148.356
C06743=1213.583,229.009,-59.974,-177.226,6.447,148.356
C06744=1213.579,229.257,-59.999,-177.223,6.449,148.355
C06745=1213.574,229.506,-60.024,-177.221,6.450,148.355
C06746=1213.570,229.755,-60.050,-177.218,6.453,148.355
C06747=1213.565,230.003,-60.076,-177.216,6.454,148.355
C06748=1213.561,230.252,-60.101,-177.213,6.456,148.354
C06749=1213.556,230.501,-60.127,-177.210,6.458,148.354
C06750=1213.551,230.749,-60.152,-177.208,6.460,148.354
C06751=1213.547,230.998,-60.177,-177.206,6.462,148.354
C06752=1213.542,231.246,-60.203,-177.203,6.464,148.353
C06753=1213.538,231.495,-60.229,-177.200,6.466,148.353
C06754=1213.534,231.744,-60.254,-177.198,6.468,148.353
C06755=1213.529,231.992,-60.280,-177.195,6.470,148.352
C06756=1213.525,232.241,-60.305,-177.193,6.472,148.352
C06757=1213.520,232.490,-60.331,-177.190,6.475,148.352
C06758=1213.515,232.738,-60.356,-177.187,6.476,148.352
C06759=1213.511,232.987,-60.382,-177.185,6.478,148.351
C06760=1213.507,233.236,-60.407,-177.182,6.480,148.351
C06761=1213.502,233.484,-60.433,-177.180,6.482,148.351
C06762=1213.498,233.733,-60.459,-177.177,6.484,148.350
C06763=1213.493,233.982,-60.485,-177.175,6.486,148.350
C06764=1213.488,234.230,-60.510,-177.172,6.488,148.350
C06765=1213.484,234.479,-60.536,-177.170,6.490,148.350
C06766=1213.480,234.728,-60.562,-177.167,6.492,148.349
C06767=1213.475,234.976,-60.588,-177.165,6.494,148.349
C06768=1213.471,235.224,-60.613,-177.162,6.496,148.349
C06769=1213.466,235.473,-60.639,-177.159,6.499,148.349
C06770=1213.462,235.722,-60.664,-177.157,6.500,148.348
C06771=1213.457,235.971,-60.690,-177.154,6.502,148.348
C06772=1213.452,236.219,-60.716,-177.152,6.504,148.348
C06773=1213.448,236.468,-60.742,-177.149,6.506,148.348
C06774=1213.444,236.717,-60.768,-177.147,6.508,148.347
C06775=1213.439,236.988,-60.795,-177.144,6.510,148.347
C06776=1213.434,237.259,-60.824,-177.141,6.513,148.347
C06777=1213.429,237.531,-60.852,-177.138,6.515,148.346
C06778=1213.425,237.802,-60.880,-177.135,6.516,148.346
C06779=1213.420,238.051,-60.907,-177.133,6.519,148.346
C06780=1213.415,238.300,-60.933,-177.130,6.521,148.346
C06781=1213.411,238.548,-60.958,-177.128,6.523,148.345
C06782=1213.406,238.797,-60.984,-177.125,6.525,148.345
C06783=1213.401,239.046,-61.010,-177.123,6.527,148.345
C06784=1213.397,239.294,-61.037,-177.120,6.529,148.345
C06785=1213.393,239.543,-61.062,-177.118,6.531,148.344
C06786=1213.388,239.791,-61.088,-177.115,6.533,148.344
C06787=1213.383,240.040,-61.114,-177.113,6.535,148.344
C06788=1213.379,240.289,-61.140,-177.110,6.538,148.344
C06789=1213.375,240.537,-61.166,-177.107,6.540,148.344
C06790=1213.371,240.786,-61.192,-177.105,6.542,148.343
C06791=1213.366,241.034,-61.218,-177.102,6.544,148.343
C06792=1213.362,241.282,-61.244,-177.100,6.545,148.343
C06793=1213.357,241.531,-61.270,-177.097,6.548,148.343
C06794=1213.352,241.780,-61.297,-177.095,6.549,148.342
C06795=1213.348,242.029,-61.322,-177.092,6.551,148.342
C06796=1213.344,242.277,-61.348,-177.089,6.554,148.342
C06797=1213.339,242.526,-61.375,-177.087,6.556,148.342
C06798=1213.335,242.775,-61.400,-177.084,6.558,148.341
C06799=1213.331,243.023,-61.427,-177.082,6.560,148.341
C06800=1213.326,243.272,-61.453,-177.079,6.562,148.341
C06801=1213.322,243.520,-61.480,-177.077,6.564,148.340
C06802=1213.317,243.769,-61.506,-177.075,6.566,148.340
C06803=1213.313,244.018,-61.532,-177.072,6.569,148.340
C06804=1213.308,244.265,-61.558,-177.069,6.571,148.340
C06805=1213.303,244.515,-61.584,-177.067,6.573,148.340
C06806=1213.299,244.763,-61.611,-177.064,6.575,148.339
C06807=1213.294,245.012,-61.637,-177.061,6.577,148.339
C06808=1213.290,245.260,-61.664,-177.059,6.579,148.339
C06809=1213.286,245.509,-61.689,-177.057,6.581,148.339
C06810=1213.281,245.757,-61.716,-177.054,6.583,148.338
C06811=1213.277,246.006,-61.742,-177.051,6.586,148.338
C06812=1213.272,246.255,-61.769,-177.049,6.587,148.338
C06813=1213.268,246.503,-61.795,-177.046,6.589,148.338
C06814=1213.263,246.751,-61.822,-177.044,6.591,148.338
C06815=1213.259,247.000,-61.847,-177.041,6.593,148.337
C06816=1213.254,247.249,-61.874,-177.039,6.595,148.337
C06817=1213.250,247.497,-61.900,-177.036,6.598,148.337
C06818=1213.245,247.746,-61.927,-177.033,6.600,148.337
C06819=1213.241,247.994,-61.954,-177.031,6.602,148.336
C06820=1213.236,248.243,-61.980,-177.029,6.604,148.336
C06821=1213.232,248.491,-62.007,-177.026,6.606,148.336
C06822=1213.227,248.740,-62.033,-177.023,6.608,148.336
C06823=1213.224,248.989,-62.059,-177.021,6.611,148.336
C06824=1213.219,249.237,-62.086,-177.018,6.613,148.335
C06825=1213.215,249.486,-62.112,-177.016,6.615,148.335
C06826=1213.210,249.734,-62.139,-177.013,6.617,148.335
C06827=1213.206,249.983,-62.166,-177.011,6.619,148.335
C06828=1213.201,250.232,-62.192,-177.009,6.621,148.334
C06829=1213.196,250.480,-62.219,-177.005,6.623,148.334
C06830=1213.193,250.728,-62.246,-177.003,6.625,148.334
C06831=1213.188,250.978,-62.272,-177.001,6.628,148.334
C06832=1213.184,251.226,-62.298,-176.998,6.629,148.333
C06833=1213.179,251.474,-62.325,-176.995,6.631,148.333
C06834=1213.174,251.723,-62.353,-176.993,6.634,148.333
C06835=1213.170,251.971,-62.379,-176.990,6.636,148.333
C06836=1213.165,252.220,-62.405,-176.988,6.638,148.333
C06837=1213.161,252.468,-62.432,-176.985,6.640,148.332
C06838=1213.157,252.717,-62.459,-176.983,6.642,148.332
C06839=1213.152,252.965,-62.486,-176.980,6.645,148.332
C06840=1213.148,253.214,-62.513,-176.977,6.647,148.332
C06841=1213.143,253.462,-62.539,-176.975,6.649,148.332
C06842=1213.139,253.711,-62.566,-176.973,6.651,148.331
C06843=1213.134,253.959,-62.593,-176.970,6.653,148.331
C06844=1213.130,254.208,-62.619,-176.967,6.656,148.331
C06845=1213.125,254.456,-62.646,-176.965,6.658,148.331
C06846=1213.121,254.705,-62.673,-176.963,6.660,148.331
C06847=1213.117,254.953,-62.700,-176.960,6.662,148.330
C06848=1213.112,255.201,-62.727,-176.958,6.664,148.330
C06849=1213.108,255.451,-62.754,-176.955,6.667,148.330
C06850=1213.104,255.699,-62.781,-176.952,6.669,148.330
C06851=1213.099,255.948,-62.807,-176.950,6.671,148.330
C06852=1213.095,256.196,-62.834,-176.947,6.673,148.329
C06853=1213.090,256.445,-62.861,-176.945,6.675,148.329
C06854=1213.085,256.693,-62.888,-176.942,6.677,148.329
C06855=1213.081,256.941,-62.915,-176.939,6.679,148.329
C06856=1213.077,257.190,-62.942,-176.937,6.682,148.328
C06857=1213.072,257.438,-62.969,-176.935,6.683,148.328
C06858=1213.068,257.688,-62.996,-176.932,6.686,148.328
C06859=1213.064,257.936,-63.024,-176.929,6.688,148.328
C06860=1213.060,258.184,-63.051,-176.927,6.690,148.328
C06861=1213.055,258.432,-63.078,-176.925,6.692,148.327
C06862=1213.050,258.681,-63.105,-176.922,6.695,148.327
C06863=1213.046,258.929,-63.132,-176.919,6.697,148.327
C06864=1213.041,259.178,-63.159,-176.917,6.699,148.327
C06865=1213.037,259.427,-63.186,-176.915,6.701,148.327
C06866=1213.033,259.675,-63.213,-176.911,6.704,148.326
C06867=1213.029,259.924,-63.240,-176.909,6.706,148.326
C06868=1213.024,260.171,-63.268,-176.907,6.708,148.326
C06869=1213.020,260.420,-63.295,-176.904,6.710,148.326
C06870=1213.015,260.668,-63.322,-176.902,6.712,148.326
C06871=1213.011,260.918,-63.349,-176.899,6.715,148.326
C06872=1213.006,261.166,-63.376,-176.897,6.717,148.325
C06873=1213.001,261.415,-63.403,-176.894,6.719,148.325
C06874=1212.997,261.663,-63.431,-176.892,6.721,148.325
C06875=1212.992,261.911,-63.458,-176.889,6.724,148.325
C06876=1212.988,262.160,-63.486,-176.886,6.726,148.325
C06877=1212.985,262.408,-63.512,-176.884,6.728,148.324
C06878=1212.980,262.656,-63.540,-176.881,6.731,148.324
C06879=1212.975,262.929,-63.570,-176.879,6.733,148.324
C06880=1212.970,263.202,-63.599,-176.876,6.736,148.324
C06881=1212.965,263.475,-63.630,-176.873,6.738,148.324
C06882=1212.960,263.748,-63.660,-176.870,6.740,148.323
C06883=1212.955,263.996,-63.687,-176.868,6.742,148.323
C06884=1212.951,264.244,-63.715,-176.865,6.744,148.323
C06885=1212.947,264.493,-63.742,-176.863,6.747,148.323
C06886=1212.943,264.741,-63.770,-176.860,6.749,148.323
C06887=1212.938,264.990,-63.797,-176.858,6.751,148.323
C06888=1212.933,265.238,-63.824,-176.855,6.754,148.322
C06889=1212.930,265.487,-63.852,-176.853,6.756,148.322
C06890=1212.925,265.735,-63.879,-176.850,6.759,148.322
C06891=1212.921,265.983,-63.907,-176.848,6.760,148.322
C06892=1212.916,266.232,-63.934,-176.845,6.763,148.322
C06893=1212.912,266.481,-63.962,-176.843,6.765,148.321
C06894=1212.908,266.729,-63.990,-176.840,6.767,148.321
C06895=1212.903,266.977,-64.017,-176.837,6.770,148.321
C06896=1212.899,267.226,-64.045,-176.835,6.772,148.321
C06897=1212.895,267.474,-64.072,-176.832,6.774,148.321
C06898=1212.890,267.722,-64.100,-176.830,6.776,148.321
C06899=1212.885,267.972,-64.128,-176.827,6.779,148.320
C06900=1212.881,268.220,-64.155,-176.825,6.781,148.320
C06901=1212.876,268.468,-64.182,-176.822,6.783,148.320
C06902=1212.872,268.716,-64.210,-176.820,6.786,148.320
C06903=1212.868,268.964,-64.238,-176.817,6.788,148.320
C06904=1212.864,269.213,-64.265,-176.815,6.790,148.320
C06905=1212.859,269.461,-64.293,-176.812,6.793,148.320
C06906=1212.854,269.710,-64.321,-176.810,6.795,148.319
C06907=1212.850,269.958,-64.349,-176.808,6.797,148.319
C06908=1212.846,270.207,-64.377,-176.805,6.799,148.319
C06909=1212.842,270.455,-64.404,-176.802,6.802,148.319
C06910=1212.837,270.703,-64.432,-176.800,6.804,148.319
C06911=1212.833,270.953,-64.460,-176.798,6.806,148.319
C06912=1212.828,271.201,-64.488,-176.794,6.809,148.318
C06913=1212.824,271.448,-64.516,-176.792,6.811,148.318
C06914=1212.820,271.697,-64.544,-176.790,6.813,148.318
C06915=1212.815,271.946,-64.571,-176.787,6.816,148.318
C06916=1212.811,272.194,-64.599,-176.785,6.818,148.318
C06917=1212.807,272.442,-64.627,-176.782,6.820,148.317
C06918=1212.802,272.691,-64.654,-176.780,6.823,148.317
C06919=1212.797,272.940,-64.683,-176.777,6.825,148.317
C06920=1212.793,273.188,-64.711,-176.775,6.827,148.317
C06921=1212.789,273.436,-64.739,-176.772,6.830,148.317
C06922=1212.785,273.684,-64.767,-176.769,6.832,148.317
C06923=1212.780,273.933,-64.794,-176.767,6.834,148.317
C06924=1212.776,274.181,-64.823,-176.765,6.837,148.317
C06925=1212.772,274.429,-64.850,-176.762,6.839,148.316
C06926=1212.767,274.678,-64.879,-176.760,6.842,148.316
C06927=1212.763,274.926,-64.907,-176.757,6.844,148.316
C06928=1212.759,275.175,-64.934,-176.755,6.846,148.316
C06929=1212.754,275.423,-64.963,-176.752,6.849,148.316
C06930=1212.750,275.672,-64.991,-176.749,6.851,148.316
C06931=1212.745,275.920,-65.019,-176.747,6.854,148.316
C06932=1212.741,276.169,-65.047,-176.745,6.855,148.315
C06933=1212.737,276.417,-65.075,-176.742,6.858,148.315
C06934=1212.732,276.665,-65.103,-176.740,6.861,148.315
C06935=1212.728,276.913,-65.132,-176.737,6.863,148.315
C06936=1212.723,277.161,-65.159,-176.734,6.866,148.315
C06937=1212.719,277.410,-65.188,-176.732,6.868,148.315
C06938=1212.715,277.658,-65.216,-176.729,6.870,148.315
C06939=1212.710,277.907,-65.245,-176.727,6.873,148.314
C06940=1212.706,278.155,-65.272,-176.725,6.875,148.314
C06941=1212.702,278.403,-65.301,-176.722,6.878,148.314
C06942=1212.698,278.652,-65.329,-176.720,6.880,148.314
C06943=1212.693,278.900,-65.357,-176.717,6.882,148.314
C06944=1212.689,279.149,-65.386,-176.714,6.885,148.314
C06945=1212.684,279.397,-65.414,-176.712,6.887,148.314
C06946=1212.680,279.646,-65.442,-176.710,6.889,148.313
C06947=1212.675,279.894,-65.470,-176.707,6.892,148.313
C06948=1212.671,280.143,-65.499,-176.705,6.894,148.313
C06949=1212.667,280.390,-65.527,-176.702,6.897,148.313
C06950=1212.662,280.639,-65.555,-176.700,6.899,148.313
C06951=1212.658,280.887,-65.584,-176.697,6.901,148.313
C06952=1212.654,281.135,-65.613,-176.694,6.904,148.313
C06953=1212.650,281.384,-65.641,-176.692,6.906,148.313
C06954=1212.645,281.632,-65.669,-176.689,6.909,148.313
C06955=1212.641,281.881,-65.697,-176.687,6.911,148.312
C06956=1212.636,282.129,-65.726,-176.685,6.913,148.312
C06957=1212.633,282.377,-65.754,-176.682,6.916,148.312
C06958=1212.627,282.625,-65.783,-176.680,6.918,148.312
C06959=1212.623,282.874,-65.812,-176.677,6.920,148.312
C06960=1212.619,283.123,-65.840,-176.675,6.923,148.312
C06961=1212.614,283.371,-65.868,-176.672,6.925,148.312
C06962=1212.611,283.619,-65.897,-176.669,6.928,148.311
C06963=1212.606,283.867,-65.925,-176.667,6.930,148.311
C06964=1212.601,284.116,-65.954,-176.665,6.933,148.311
C06965=1212.598,284.364,-65.983,-176.662,6.936,148.311
C06966=1212.593,284.612,-66.011,-176.660,6.937,148.311
C06967=1212.588,284.861,-66.040,-176.657,6.940,148.311
C06968=1212.585,285.109,-66.069,-176.655,6.943,148.311
C06969=1212.580,285.357,-66.097,-176.653,6.945,148.311
C06970=1212.575,285.606,-66.126,-176.650,6.948,148.311
C06971=1212.571,285.853,-66.154,-176.648,6.950,148.311
C06972=1212.566,286.102,-66.183,-176.645,6.953,148.310
C06973=1212.562,286.351,-66.212,-176.642,6.955,148.310
C06974=1212.558,286.598,-66.240,-176.640,6.958,148.310
C06975=1212.553,286.847,-66.269,-176.637,6.960,148.310
C06976=1212.549,287.095,-66.299,-176.635,6.962,148.310
C06977=1212.545,287.343,-66.326,-176.632,6.965,148.310
C06978=1212.541,287.591,-66.356,-176.630,6.967,148.310
C06979=1212.536,287.840,-66.385,-176.627,6.970,148.310
C06980=1212.532,288.089,-66.413,-176.625,6.972,148.310
C06981=1212.528,288.336,-66.442,-176.623,6.974,148.310
C06982=1212.523,288.585,-66.471,-176.620,6.977,148.309
C06983=1212.519,288.859,-66.503,-176.617,6.980,148.309
C06984=1212.514,289.133,-66.535,-176.615,6.982,148.309
C06985=1212.509,289.408,-66.566,-176.612,6.985,148.309
C06986=1212.504,289.682,-66.599,-176.609,6.988,148.309
C06987=1212.500,289.930,-66.627,-176.607,6.990,148.309
C06988=1212.495,290.178,-66.656,-176.604,6.993,148.309
C06989=1212.491,290.427,-66.685,-176.602,6.995,148.309
C06990=1212.487,290.675,-66.715,-176.599,6.998,148.309
C06991=1212.482,290.924,-66.743,-176.597,7.000,148.309
C06992=1212.478,291.171,-66.772,-176.594,7.004,148.309
C06993=1212.474,291.420,-66.801,-176.592,7.006,148.308
C06994=1212.470,291.668,-66.830,-176.589,7.008,148.308
C06995=1212.465,291.917,-66.859,-176.587,7.011,148.308
C06996=1212.461,292.165,-66.889,-176.585,7.013,148.308
C06997=1212.456,292.413,-66.917,-176.582,7.016,148.308
C06998=1212.452,292.661,-66.947,-176.580,7.018,148.308
C06999=1212.448,292.910,-66.976,-176.577,7.021,148.308
C07000=1212.444,293.158,-67.005,-176.575,7.023,148.308
C07001=1212.439,293.406,-67.033,-176.572,7.026,148.308
C07002=1212.435,293.654,-67.063,-176.570,7.028,148.308
C07003=1212.431,293.902,-67.092,-176.567,7.031,148.308
C07004=1212.427,294.151,-67.122,-176.565,7.033,148.308
C07005=1212.422,294.400,-67.151,-176.563,7.036,148.307
C07006=1212.417,294.647,-67.180,-176.560,7.038,148.307
C07007=1212.413,294.895,-67.209,-176.558,7.041,148.307
C07008=1212.409,295.144,-67.239,-176.555,7.044,148.307
C07009=1212.405,295.392,-67.268,-176.553,7.046,148.307
C07010=1212.400,295.641,-67.297,-176.550,7.049,148.307
C07011=1212.396,295.889,-67.326,-176.548,7.051,148.307
C07012=1212.392,296.137,-67.356,-176.545,7.054,148.307
C07013=1212.387,296.385,-67.385,-176.543,7.056,148.307
C07014=1212.383,296.633,-67.414,-176.540,7.059,148.307
C07015=1212.379,296.881,-67.444,-176.538,7.061,148.307
C07016=1212.375,297.130,-67.473,-176.535,7.064,148.307
C07017=1212.370,297.378,-67.503,-176.533,7.066,148.307
C07018=1212.366,297.626,-67.532,-176.531,7.069,148.307
C07019=1212.362,297.875,-67.561,-176.528,7.072,148.307
C07020=1212.357,298.123,-67.590,-176.526,7.074,148.306
C07021=1212.353,298.371,-67.619,-176.524,7.077,148.306
C07022=1212.349,298.619,-67.649,-176.522,7.079,148.306
C07023=1212.344,298.868,-67.678,-176.518,7.082,148.306
C07024=1212.340,299.116,-67.708,-176.516,7.084,148.306
C07025=1212.336,299.364,-67.737,-176.514,7.087,148.306
C07026=1212.332,299.612,-67.767,-176.511,7.089,148.306
C07027=1212.327,299.861,-67.797,-176.509,7.092,148.306
C07028=1212.323,300.109,-67.827,-176.507,7.094,148.306
C07029=1212.319,300.357,-67.856,-176.504,7.098,148.306
C07030=1212.315,300.605,-67.886,-176.502,7.100,148.306
C07031=1212.310,300.853,-67.915,-176.499,7.103,148.306
C07032=1212.306,301.101,-67.944,-176.497,7.105,148.306
C07033=1212.302,301.349,-67.974,-176.494,7.108,148.306
C07034=1212.297,301.598,-68.004,-176.492,7.110,148.306
C07035=1212.293,301.846,-68.033,-176.490,7.113,148.306
C07036=1212.288,302.094,-68.063,-176.487,7.115,148.306
C07037=1212.284,302.342,-68.093,-176.485,7.118,148.306
C07038=1212.280,302.590,-68.122,-176.483,7.121,148.306
C07039=1212.276,302.838,-68.152,-176.480,7.124,148.306
C07040=1212.271,303.087,-68.182,-176.478,7.126,148.305
C07041=1212.267,303.335,-68.211,-176.475,7.129,148.305
C07042=1212.263,303.583,-68.241,-176.473,7.131,148.305
C07043=1212.259,303.831,-68.271,-176.470,7.134,148.305
C07044=1212.254,304.080,-68.301,-176.468,7.136,148.305
C07045=1212.250,304.328,-68.330,-176.466,7.139,148.305
C07046=1212.246,304.576,-68.360,-176.463,7.142,148.305
C07047=1212.242,304.824,-68.390,-176.461,7.145,148.305
C07048=1212.237,305.073,-68.420,-176.459,7.147,148.305
C07049=1212.233,305.321,-68.449,-176.456,7.150,148.305
C07050=1212.229,305.568,-68.480,-176.454,7.152,148.305
C07051=1212.224,305.817,-68.510,-176.451,7.155,148.305
C07052=1212.220,306.065,-68.539,-176.449,7.157,148.305
C07053=1212.216,306.313,-68.569,-176.446,7.160,148.305
C07054=1212.211,306.562,-68.599,-176.444,7.163,148.305
C07055=1212.207,306.810,-68.629,-176.442,7.166,148.305
C07056=1212.203,307.057,-68.659,-176.439,7.168,148.305
C07057=1212.198,307.306,-68.689,-176.437,7.171,148.305
C07058=1212.194,307.554,-68.719,-176.435,7.173,148.305
C07059=1212.190,307.802,-68.749,-176.432,7.176,148.305
C07060=1212.185,308.050,-68.779,-176.430,7.178,148.305
C07061=1212.182,308.299,-68.809,-176.427,7.181,148.305
C07062=1212.177,308.547,-68.839,-176.425,7.184,148.305
C07063=1212.173,308.795,-68.869,-176.422,7.187,148.305
C07064=1212.169,309.043,-68.899,-176.420,7.189,148.305
C07065=1212.164,309.291,-68.930,-176.418,7.192,148.305
C07066=1212.160,309.540,-68.959,-176.416,7.194,148.305
C07067=1212.156,309.787,-68.989,-176.413,7.197,148.305
C07068=1212.151,310.036,-69.019,-176.411,7.200,148.305
C07069=1212.147,310.283,-69.049,-176.408,7.203,148.305
C07070=1212.143,310.531,-69.080,-176.406,7.205,148.305
C07071=1212.138,310.780,-69.110,-176.404,7.208,148.305
C07072=1212.134,311.028,-69.141,-176.402,7.210,148.305
C07073=1212.130,311.277,-69.170,-176.399,7.213,148.305
C07074=1212.126,311.525,-69.201,-176.397,7.216,148.305
C07075=1212.122,311.772,-69.231,-176.395,7.219,148.305
C07076=1212.117,312.021,-69.261,-176.392,7.222,148.305
C07077=1212.113,312.268,-69.291,-176.390,7.224,148.305
C07078=1212.108,312.517,-69.321,-176.387,7.227,148.305
C07079=1212.105,312.765,-69.352,-176.385,7.229,148.305
C07080=1212.100,313.013,-69.383,-176.382,7.232,148.305
C07081=1212.096,313.262,-69.412,-176.381,7.235,148.305
C07082=1212.091,313.510,-69.443,-176.378,7.238,148.305
C07083=1212.087,313.757,-69.473,-176.376,7.240,148.305
C07084=1212.083,314.005,-69.504,-176.373,7.243,148.305
C07085=1212.079,314.254,-69.534,-176.371,7.245,148.305
C07086=1212.075,314.502,-69.564,-176.368,7.248,148.305
C07087=1212.070,314.778,-69.599,-176.366,7.252,148.305
C07088=1212.065,315.054,-69.632,-176.364,7.255,148.305
C07089=1212.061,315.330,-69.666,-176.361,7.258,148.305
C07090=1212.056,315.606,-69.700,-176.358,7.261,148.305
C07091=1212.051,315.854,-69.730,-176.356,7.263,148.305
C07092=1212.047,316.102,-69.761,-176.353,7.266,148.305
C07093=1212.043,316.350,-69.792,-176.352,7.268,148.305
C07094=1212.039,316.598,-69.822,-176.349,7.272,148.305
C07095=1212.035,316.846,-69.853,-176.347,7.274,148.305
C07096=1212.030,317.095,-69.883,-176.344,7.277,148.305
C07097=1212.026,317.343,-69.914,-176.343,7.279,148.305
C07098=1212.022,317.591,-69.944,-176.340,7.282,148.305
C07099=1212.017,317.839,-69.975,-176.338,7.285,148.305
C07100=1212.013,318.087,-70.005,-176.335,7.288,148.305
C07101=1212.009,318.335,-70.036,-176.333,7.291,148.305
C07102=1212.005,318.583,-70.067,-176.331,7.293,148.305
C07103=1212.000,318.831,-70.098,-176.328,7.296,148.305
C07104=1211.996,319.079,-70.128,-176.326,7.298,148.305
C07105=1211.992,319.327,-70.159,-176.324,7.302,148.305
C07106=1211.988,319.575,-70.190,-176.322,7.304,148.305
C07107=1211.984,319.823,-70.220,-176.319,7.307,148.305
C07108=1211.980,320.072,-70.251,-176.317,7.309,148.305
C07109=1211.975,320.320,-70.282,-176.315,7.312,148.306
C07110=1211.971,320.568,-70.312,-176.313,7.315,148.306
C07111=1211.967,320.815,-70.343,-176.310,7.318,148.306
C07112=1211.963,321.064,-70.374,-176.308,7.320,148.306
C07113=1211.958,321.312,-70.404,-176.306,7.323,148.306
C07114=1211.953,321.560,-70.435,-176.303,7.326,148.306
C07115=1211.949,321.808,-70.466,-176.301,7.329,148.306
C07116=1211.946,322.056,-70.497,-176.299,7.332,148.306
C07117=1211.941,322.303,-70.528,-176.296,7.334,148.306
C07118=1211.937,322.552,-70.559,-176.294,7.337,148.306
C07119=1211.933,322.800,-70.590,-176.292,7.340,148.306
C07120=1211.928,323.048,-70.621,-176.289,7.343,148.306
C07121=1211.925,323.296,-70.651,-176.288,7.345,148.306
C07122=1211.920,323.544,-70.682,-176.285,7.348,148.306
C07123=1211.916,323.792,-70.714,-176.284,7.351,148.306
C07124=1211.912,324.040,-70.745,-176.281,7.354,148.306
C07125=1211.907,324.288,-70.775,-176.278,7.357,148.306
C07126=1211.903,324.537,-70.806,-176.277,7.359,148.306
C07127=1211.899,324.785,-70.837,-176.274,7.362,148.306
C07128=1211.895,325.032,-70.868,-176.272,7.365,148.307
C07129=1211.891,325.281,-70.899,-176.270,7.368,148.307
C07130=1211.886,325.529,-70.930,-176.267,7.370,148.307
C07131=1211.883,325.777,-70.962,-176.265,7.374,148.307
C07132=1211.878,326.025,-70.993,-176.263,7.376,148.307
C07133=1211.873,326.273,-71.023,-176.261,7.379,148.307
C07134=1211.870,326.521,-71.055,-176.258,7.382,148.307
C07135=1211.865,326.769,-71.086,-176.257,7.385,148.307
C07136=1211.861,327.017,-71.117,-176.254,7.388,148.307
C07137=1211.857,327.265,-71.149,-176.252,7.390,148.307
C07138=1211.853,327.513,-71.180,-176.250,7.393,148.307
C07139=1211.848,327.761,-71.210,-176.247,7.395,148.307
C07140=1211.844,328.008,-71.242,-176.245,7.399,148.308
C07141=1211.840,328.257,-71.273,-176.243,7.401,148.307
C07142=1211.836,328.504,-71.305,-176.241,7.404,148.308
C07143=1211.832,328.753,-71.336,-176.239,7.407,148.308
C07144=1211.827,329.001,-71.366,-176.237,7.410,148.308
C07145=1211.823,329.249,-71.398,-176.234,7.413,148.308
C07146=1211.819,329.497,-71.429,-176.232,7.415,148.308
C07147=1211.815,329.745,-71.461,-176.230,7.419,148.308
C07148=1211.810,329.993,-71.492,-176.228,7.421,148.308
C07149=1211.807,330.241,-71.524,-176.225,7.424,148.308
C07150=1211.802,330.489,-71.554,-176.224,7.427,148.308
C07151=1211.798,330.737,-71.586,-176.221,7.430,148.308
C07152=1211.794,330.985,-71.617,-176.219,7.432,148.309
C07153=1211.790,331.233,-71.649,-176.217,7.435,148.309
C07154=1211.786,331.480,-71.680,-176.215,7.438,148.309
C07155=1211.782,331.729,-71.711,-176.213,7.441,148.309
C07156=1211.777,331.976,-71.743,-176.210,7.444,148.309
C07157=1211.773,332.225,-71.774,-176.208,7.447,148.309
C07158=1211.768,332.473,-71.806,-176.206,7.450,148.309
C07159=1211.765,332.721,-71.838,-176.204,7.452,148.309
C07160=1211.760,332.969,-71.869,-176.202,7.456,148.310
C07161=1211.756,333.217,-71.900,-176.200,7.458,148.310
C07162=1211.752,333.465,-71.931,-176.198,7.461,148.310
C07163=1211.748,333.713,-71.963,-176.196,7.463,148.310
C07164=1211.744,333.960,-71.995,-176.193,7.467,148.310
C07165=1211.739,334.209,-72.026,-176.192,7.469,148.310
C07166=1211.735,334.456,-72.058,-176.189,7.472,148.310
C07167=1211.731,334.704,-72.090,-176.187,7.476,148.310
C07168=1211.727,334.952,-72.121,-176.185,7.478,148.311
C07169=1211.722,335.200,-72.152,-176.182,7.481,148.311
C07170=1211.718,335.449,-72.185,-176.181,7.484,148.311
C07171=1211.714,335.696,-72.216,-176.179,7.487,148.311
C07172=1211.710,335.944,-72.248,-176.177,7.489,148.311
C07173=1211.705,336.192,-72.279,-176.174,7.493,148.311
C07174=1211.702,336.440,-72.311,-176.173,7.495,148.311
C07175=1211.697,336.689,-72.343,-176.170,7.498,148.311
C07176=1211.693,336.936,-72.375,-176.168,7.501,148.311
C07177=1211.689,337.184,-72.406,-176.166,7.504,148.312
C07178=1211.685,337.431,-72.438,-176.164,7.506,148.312
C07179=1211.680,337.680,-72.470,-176.162,7.509,148.312
C07180=1211.676,337.928,-72.501,-176.160,7.513,148.312
C07181=1211.672,338.176,-72.533,-176.158,7.515,148.312
C07182=1211.668,338.424,-72.565,-176.155,7.518,148.312
C07183=1211.663,338.671,-72.597,-176.154,7.521,148.312
C07184=1211.660,338.919,-72.629,-176.151,7.524,148.313
C07185=1211.655,339.168,-72.661,-176.150,7.527,148.313
C07186=1211.651,339.415,-72.693,-176.147,7.530,148.313
C07187=1211.647,339.663,-72.724,-176.145,7.532,148.313
C07188=1211.644,339.911,-72.756,-176.143,7.536,148.313
C07189=1211.639,340.159,-72.788,-176.142,7.538,148.313
C07190=1211.635,340.407,-72.820,-176.139,7.542,148.314
C07191=1211.629,340.685,-72.856,-176.137,7.545,148.314
C07192=1211.625,340.963,-72.891,-176.135,7.548,148.314
C07193=1211.621,341.241,-72.928,-176.132,7.551,148.314
C07194=1211.615,341.520,-72.963,-176.130,7.555,148.314
C07195=1211.612,341.768,-72.995,-176.128,7.557,148.315
C07196=1211.607,342.015,-73.027,-176.126,7.560,148.315
C07197=1211.603,342.263,-73.060,-176.124,7.563,148.315
C07198=1211.599,342.511,-73.092,-176.122,7.566,148.315
C07199=1211.594,342.759,-73.124,-176.120,7.569,148.315
C07200=1211.591,343.007,-73.156,-176.118,7.572,148.315
C07201=1211.586,343.255,-73.188,-176.116,7.574,148.316
C07202=1211.582,343.502,-73.220,-176.114,7.578,148.316
C07203=1211.578,343.750,-73.251,-176.113,7.580,148.316
C07204=1211.574,343.999,-73.284,-176.110,7.583,148.316
C07205=1211.570,344.247,-73.316,-176.108,7.586,148.316
C07206=1211.565,344.494,-73.348,-176.106,7.589,148.316
C07207=1211.562,344.742,-73.380,-176.104,7.592,148.316
C07208=1211.557,344.990,-73.413,-176.102,7.595,148.317
C07209=1211.553,345.237,-73.444,-176.100,7.598,148.317
C07210=1211.548,345.486,-73.477,-176.098,7.601,148.317
C07211=1211.545,345.733,-73.509,-176.096,7.604,148.317
C07212=1211.541,345.982,-73.542,-176.095,7.607,148.318
C07213=1211.536,346.229,-73.573,-176.092,7.610,148.318
C07214=1211.532,346.477,-73.606,-176.091,7.613,148.318
C07215=1211.528,346.725,-73.638,-176.088,7.616,148.318
C07216=1211.524,346.973,-73.671,-176.087,7.619,148.318
C07217=1211.520,347.221,-73.703,-176.085,7.622,148.319
C07218=1211.515,347.469,-73.734,-176.083,7.624,148.319
C07219=1211.511,347.716,-73.768,-176.081,7.628,148.319
C07220=1211.507,347.965,-73.799,-176.079,7.630,148.319
C07221=1211.503,348.213,-73.832,-176.077,7.634,148.319
C07222=1211.498,348.460,-73.865,-176.075,7.636,148.320
C07223=1211.495,348.708,-73.897,-176.073,7.639,148.320
C07224=1211.490,348.956,-73.930,-176.071,7.642,148.320
C07225=1211.487,349.204,-73.962,-176.069,7.645,148.320
C07226=1211.482,349.452,-73.994,-176.068,7.648,148.320
C07227=1211.478,349.699,-74.027,-176.065,7.651,148.321
C07228=1211.474,349.947,-74.059,-176.064,7.654,148.321
C07229=1211.470,350.195,-74.092,-176.061,7.657,148.321
C07230=1211.466,350.443,-74.124,-176.060,7.660,148.321
C07231=1211.462,350.691,-74.156,-176.058,7.663,148.322
C07232=1211.457,350.939,-74.189,-176.056,7.666,148.322
C07233=1211.453,351.186,-74.221,-176.054,7.669,148.322
C07234=1211.449,351.434,-74.254,-176.053,7.672,148.322
C07235=1211.444,351.682,-74.286,-176.051,7.674,148.322
C07236=1211.440,351.930,-74.319,-176.049,7.677,148.323
C07237=1211.437,352.178,-74.351,-176.048,7.680,148.323
C07238=1211.432,352.426,-74.384,-176.045,7.684,148.323
C07239=1211.428,352.674,-74.417,-176.044,7.686,148.323
C07240=1211.424,352.921,-74.449,-176.041,7.690,148.324
C07241=1211.420,353.169,-74.482,-176.040,7.692,148.324
C07242=1211.415,353.417,-74.515,-176.038,7.695,148.324
C07243=1211.411,353.665,-74.548,-176.036,7.698,148.324
C07244=1211.408,353.913,-74.580,-176.034,7.702,148.325
C07245=1211.403,354.161,-74.613,-176.033,7.704,148.325
C07246=1211.399,354.409,-74.645,-176.030,7.707,148.325
C07247=1211.395,354.657,-74.678,-176.029,7.710,148.325
C07248=1211.392,354.904,-74.711,-176.027,7.714,148.326
C07249=1211.386,355.152,-74.743,-176.025,7.716,148.326
C07250=1211.382,355.399,-74.776,-176.023,7.719,148.326
C07251=1211.378,355.647,-74.809,-176.022,7.722,148.327
C07252=1211.374,355.895,-74.841,-176.020,7.725,148.327
C07253=1211.370,356.143,-74.874,-176.018,7.728,148.327
C07254=1211.366,356.391,-74.908,-176.017,7.731,148.327
C07255=1211.362,356.639,-74.940,-176.015,7.734,148.328
C07256=1211.358,356.887,-74.973,-176.013,7.737,148.328
C07257=1211.353,357.134,-75.006,-176.011,7.740,148.328
C07258=1211.350,357.382,-75.039,-176.010,7.743,148.328
C07259=1211.346,357.630,-75.071,-176.007,7.746,148.329
C07260=1211.341,357.878,-75.104,-176.006,7.749,148.329
C07261=1211.337,358.126,-75.138,-176.005,7.752,148.329
C07262=1211.333,358.373,-75.171,-176.002,7.755,148.329
C07263=1211.329,358.621,-75.204,-176.001,7.758,148.330
C07264=1211.325,358.869,-75.236,-175.999,7.761,148.330
C07265=1211.321,359.117,-75.269,-175.998,7.764,148.330
C07266=1211.317,359.365,-75.302,-175.996,7.767,148.331
C07267=1211.313,359.612,-75.335,-175.994,7.770,148.331
C07268=1211.309,359.860,-75.368,-175.993,7.773,148.331
C07269=1211.305,360.108,-75.402,-175.990,7.776,148.331
C07270=1211.300,360.356,-75.434,-175.989,7.779,148.332
C07271=1211.296,360.604,-75.467,-175.987,7.782,148.332
C07272=1211.292,360.852,-75.500,-175.986,7.785,148.332
C07273=1211.288,361.099,-75.533,-175.984,7.787,148.333
C07274=1211.284,361.347,-75.567,-175.983,7.791,148.333
C07275=1211.280,361.595,-75.600,-175.981,7.794,148.333
C07276=1211.275,361.843,-75.633,-175.979,7.797,148.334
C07277=1211.272,362.090,-75.665,-175.977,7.800,148.334
C07278=1211.268,362.338,-75.699,-175.976,7.803,148.334
C07279=1211.264,362.585,-75.732,-175.974,7.806,148.335
C07280=1211.260,362.833,-75.765,-175.973,7.809,148.335
C07281=1211.255,363.081,-75.798,-175.971,7.812,148.335
C07282=1211.251,363.329,-75.831,-175.969,7.815,148.336
C07283=1211.247,363.576,-75.864,-175.968,7.818,148.336
C07284=1211.243,363.824,-75.898,-175.966,7.821,148.336
C07285=1211.239,364.072,-75.931,-175.965,7.824,148.337
C07286=1211.235,364.320,-75.964,-175.963,7.826,148.337
C07287=1211.231,364.567,-75.997,-175.961,7.830,148.337
C07288=1211.226,364.815,-76.030,-175.960,7.833,148.338
C07289=1211.222,365.063,-76.063,-175.959,7.835,148.338
C07290=1211.217,365.311,-76.097,-175.957,7.839,148.338
C07291=1211.213,365.558,-76.130,-175.956,7.842,148.339
C07292=1211.209,365.806,-76.163,-175.954,7.844,148.339
C07293=1211.206,366.055,-76.197,-175.952,7.848,148.339
C07294=1211.202,366.302,-76.231,-175.951,7.851,148.340
C07295=1211.197,366.582,-76.268,-175.949,7.855,148.340
C07296=1211.193,366.862,-76.306,-175.948,7.857,148.340
C07297=1211.188,367.142,-76.344,-175.946,7.861,148.341
C07298=1211.184,367.422,-76.382,-175.944,7.864,148.341
C07299=1211.179,367.670,-76.415,-175.943,7.867,148.342
C07300=1211.175,367.918,-76.448,-175.942,7.870,148.342
C07301=1211.171,368.166,-76.481,-175.940,7.873,148.342
C07302=1211.166,368.414,-76.515,-175.938,7.876,148.343
C07303=1211.162,368.661,-76.548,-175.937,7.879,148.343
C07304=1211.158,368.908,-76.582,-175.936,7.882,148.343
C07305=1211.155,369.157,-76.615,-175.934,7.885,148.344
C07306=1211.151,369.405,-76.648,-175.933,7.888,148.344
C07307=1211.147,369.652,-76.682,-175.931,7.891,148.344
C07308=1211.142,369.900,-76.716,-175.930,7.894,148.345
C07309=1211.138,370.148,-76.749,-175.928,7.897,148.345
C07310=1211.134,370.395,-76.782,-175.927,7.900,148.346
C07311=1211.130,370.642,-76.816,-175.926,7.903,148.346
C07312=1211.126,370.891,-76.850,-175.925,7.906,148.346
C07313=1211.122,371.139,-76.883,-175.924,7.908,148.347
C07314=1211.118,371.386,-76.917,-175.922,7.912,148.347
